(* Structure page *)
	T_ConfigPage:ST_CONFIGPAGE;
	wMaskBtPanelLeft: WORD;
	wMaskBtPanelRight: WORD;
	wMaskFunctionPanel: WORD;
	RisingEdgeProcessDone: R_TRIG;
	xStopImmediatly: BOOL;
	RisingEdgeProcessError: R_TRIG;
	RisingEdgeResetProcess: R_TRIG;
	RisingEdgeExecuteProcess: R_TRIG;
	RisingEdgeActionNotReady: R_TRIG;
	FallingEdgeActionNotReady: F_TRIG;
	RisingEdgeActionDone: R_TRIG;
	xBlockConfirmMessage: BOOL;
	RisingEdgeActionError: R_TRIG;
	RisingEdgeResetAction: R_TRIG;
	xSlowFast: BOOL;
	iSelectedAxis: INT;
	xSlowFastJogToolRotation: BOOL;
	xSlowFastJogToolFeeder: BOOL;
	xSlowFastJogGrindFeeder: BOOL;
	xToggleAxisPower: BOOL;
	xResetAxis: BOOL;
	xUpdateProfileList: BOOL;
	jj: INT;
	RisingEdgePtrProfileListUpDown: R_TRIG;
	iPointerListProfile: INT;
	iActualActiveProfile: INT;
	xAction_CopyProfileToProcess: BOOL;
	xProfileFileNotFound: BOOL;
	iToLoadProfileNr: INT;
	sToLoadProfileName: STRING;
	sTmpDynamicText: STRING;
	xAction_LoadProfileToProcessImage: BOOL;
	xAction_SaveNovRAM: BOOL;
	xActionDeleteProfile: BOOL;
	TimerONTmp: TON;
	iStepActionNovRam: INT;
	xAction_SaveProfileToFile: BOOL;
	iTmp: INT;
	sTmp: STRING;
	sTmp_2: STRING;
	RisingEdgeTimeOut: R_TRIG;
	fbCompareProfileProcessValue:FB_COMPAREPROFILEPROCESSVALUE;
	FailingEdgeGeometryManagement: F_TRIG;
	FailingEdgePrisma: F_TRIG;
	rCalcMinMaxToolDia: REAL;
	xResetParaListValue: BOOL;
	xActivateStationFunction: BOOL;
	iTmpStationFunctionNr: INT;
	xFirstReadInit: BOOL;
	xFirstReadReset: BOOL;
	xMicroRodActive: BOOL;
	FBCalcTorqueToolLeft: FB_CALC_TORQUE;
	FBCalcTorqueToolCenter: FB_CALC_TORQUE;
	FBCalcTorqueToolRight: FB_CALC_TORQUE;
	xTmpStopAxis: BOOL;
	RisingEdgeStartButton: R_TRIG;
	dwPageNrProcessStart: DWORD;
	FallingEdgeStartButton: F_TRIG;
	RisingEdgeStopButton: R_TRIG;
	FallingEdgeStopButton: F_TRIG;
	xToggleCylinderState: BOOL;
	dwTmpActualPage: DWORD;
	xUpdateErrorList: BOOL;
	RisingEdgeErrorList: R_TRIG;
	xParameterSavedErrorList: BOOL;
	xDeleteErrorList: BOOL;
	FBQVisErrorList: FBQVIS_ERROR_LIST;
	FBSetErrorList:FB_SETERRORLIST;
	xProcessMachine: BOOL;
	xProcessStation: BOOL;
	iStepProcess: INT;
	xStepProcessDone: BOOL;
	xStopProcess: BOOL;
	xAction_StopCycle: BOOL;
	xWaitStopEnd: BOOL;
	xWaitStopCycleEnd: BOOL;
	iStepWaitStopEnd: INT;
	xActionProcStation: BOOL;
	xActionProcMachine: BOOL;
	RisingEdgeKeySwitch1: R_TRIG;
	FailingEdgeKeySwitch1: F_TRIG;
	TimerDisplayMessage: TON;
	RisingEdgeReleaseWarning: R_TRIG;
	rCalcPrismaFactor: REAL;
	xFirstReadParaList: BOOL;
	iTmpSelectParaList: INT;
	xAction_SaveNovRAMWithoutConfirm: BOOL;
	diErrorNr: DINT;
	FBErrorMessage : FB_ErrorMessage;
	fbQvisClearError:FBQVIS_CLEARERROR;
	xResetError: BOOL;
	TONTimeWaitMsg: TON;
	xCheckQuitError: BOOL;
	bStateMachine: BYTE;
	xSetStateMachine: BOOL;
	iSelectAxisToolRotation: INT;
	rAutoTimeTotal: REAL;
	rToolRotationSpeed: REAL;
	iAutoProcess: INT;
	xBlockGrindFeederActivation: BOOL;
	xToolFeederMoveStartPos: BOOL;
	xToggleAllAxisPower: BOOL;
	FBCalcProcessTime: FB_CALCPROCESSTIME;
	xReferenceAxis: BOOL;
	xTeachPosition: BOOL;
	xCalcAngleRefIndex: BOOL;
	uiToolLeftZeroTorque: UINT;
	uiToolCenterZeroTorque: UINT;
	uiToolRightZeroTorque: UINT;
	xSetCalculToolRotTorque: BOOL;
	rActualToolFeederPosition: REAL;
	xReadActualToolFeedPos: BOOL;
	xReadActualToolFeedPos1: BOOL;
	rActualToolFeederPosition1: REAL;
	rToolTotalLength: REAL;
	xCalcFirstTime: BOOL;
	xFirstReadParaList1: BOOL;
	iTmpSelectParaList1: INT;
	xTmpTeach: BOOL;
	wTmpActivBtRight: WORD;
	xOverlayGrindFeedSetPlung: BOOL;
	xOpenMessageBox: BOOL;
	lrActualGrindFeedPosition: LREAL;
	lrToWriteGrindFeedPosition: LREAL;
	xCalcAgainProcTime: BOOL;
	xToolFeederMoveLoadPos: BOOL;
	xWarmUp:BOOL;
	iSelectedCylinder: INT;
	xWarmUpMessage: BOOL;
	xWarmUpMessageActiv: BOOL;
	xWarmUpMessageDone: BOOL;
END_VAR
(****************************************************************************************************************************************************)
(******    This Functionblock manage the hole visualisation, it is the interface from the QVis and the control application          *******)
(****************************************************************************************************************************************************)
	IF NOT(xFirstRead) THEN
		xFirstRead:=TRUE;
		T_Visu.ptrT_ExchgParam:=ADR(T_ExchgParam);
	END_IF;
	RisingEdgeActiv(CLK:=T_Visu.T_CtrleVisu.xActive);
	IF RisingEdgeActiv.Q THEN
		(* call functionblock init. *)
		fbQvisInitPage(T_Visu:=T_Visu);
		(* Init. variable for visualisation action *)
		T_Visu.T_CtrleAction.xDone:=TRUE;
		T_Visu.T_CtrleAction.xExecute:=FALSE;
		T_Visu.T_CtrleAction.xNotReady:=FALSE;
		T_Visu.T_CtrleAction.xErr:=FALSE;
		T_Visu.T_CtrleAction.udiErrorID:=0;
		T_Visu.T_CtrleVisu.xDone:=FALSE;
		T_Visu.ptrT_ExchgParam:=ADR(T_ExchgParam);
		wNormalLayerActivTask:=1;
		wSpecialLayerGeneralActivTask:=1;
		wSpecialLayerToolRotActivTask:=1;
		wSpecialLayerWireFeedActivTask:=1;
		wSpecialLayerGrindAxisActivTask:=1;
		wNormalLayerActivPage:=10;
		wSpecialLayerGeneralActivPage:=110;
		wSpecialLayerToolRotActivPage:=210;
		wSpecialLayerWireFeedActivPage:=310;
		wSpecialLayerGrindAxisActivPage:=410;
		T_Visu.ptrT_ExchgParam^.T_TouchScreenNavPanel.wState:=1;
		wStandardPageNr:=10;
		T_Visu.ptrT_ExchgParam^.T_Visu.T_Level.iPwSystem:=999;
		wTmpNormalLayerActivTask:=1;
		wTmpSpecialLayerGeneralActivTask:=1;
		wTmpSpecialLayerToolRotActivTask:=1;
		wTmpSpecialLayerWireFeedActivTask:=1;
		wTmpSpecialLayerGrindAxisActivTask:=1;
		FOR ii:=1 TO 6 DO
			awNormalLayerActivPage[ii]:=wStandardPageNr;
			wStandardPageNr:=wStandardPageNr + 10;
		END_FOR;
		wStandardPageNr:=110;
		FOR ii:=1 TO 6 DO
			awSpecialLayerGeneralActivPage[ii]:=wStandardPageNr;
			wStandardPageNr:=wStandardPageNr + 10;
		END_FOR;
		wStandardPageNr:=210;
		FOR ii:=1 TO 6 DO
			awSpecialLayerToolRotActivPage[ii]:=wStandardPageNr;
			wStandardPageNr:=wStandardPageNr + 10;
		END_FOR;
		wStandardPageNr:=310;
		FOR ii:=1 TO 6 DO
			awSpecialLayerWireFeedActivPage[ii]:=wStandardPageNr;
			wStandardPageNr:=wStandardPageNr + 10;
		END_FOR;
		wStandardPageNr:=410;
		FOR ii:=1 TO 6 DO
			awSpecialLayerGrindAxisActivPage[ii]:=wStandardPageNr;
			wStandardPageNr:=wStandardPageNr + 10;
		END_FOR;
		IF NOT(xFirstReadInit) THEN
			xFirstReadInit:=TRUE;
			T_Visu.T_PlcParam.dwSetNewPage:=1001;
		ELSE
			T_Visu.T_PlcParam.dwSetNewPage:=0;
		END_IF;
		T_Visu.T_PlcParam.dwActualPage:=0;
		T_Visu.T_PlcParam.dwPreviousPage:=0;
		iPointerListProfile:=1;
		iActualActiveProfile:=-1;
		TimerAction(IN:=FALSE);
		(* Init FB *)
		fbQvisClearError(	xExecute:=FALSE,
						iError:=0,
						T_Message:=T_ExchgParam.T_Visu.T_Message,
						T_Station:=T_Station,
						T_Process:=T_Process,
						T_NovRAM:=T_NovRAM,
						T_Profile:=T_Profile,
						T_HDD:=T_HDD,
						xDone=>T_Visu.T_CtrleAction.xDone,
						xNotReady=>T_Visu.T_CtrleAction.xNotReady,
						xErr=>T_Visu.T_CtrleAction.xErr,
						udiErrorID=>T_Visu.T_CtrleAction.udiErrorID);
		T_Visu.ptrT_ExchgParam^.T_Cylinder.iSelectToolTensionForce:=1;	(* For starting the machine set always the process force for the ToolTension *)
		ptrTeachINAxis:=ADR(T_Station.THardware.TAxisToolLeft);
	END_IF;

	IF NOT(T_Visu.T_CtrleVisu.xActive) THEN
		RETURN;
	END_IF;

(* waiting for reset *)
	RisingEdgeReset(CLK:=T_Visu.T_CtrleVisu.xReset);
	IF RisingEdgeReset.Q THEN
		(* Init. structure *)
		T_Visu.T_CtrleVisu.xDone:=FALSE;
		T_Visu.T_CtrleVisu.iFunction:=0;
		T_Visu.T_CtrleVisu.xErr:=FALSE;
		T_Visu.T_CtrleVisu.udiErrorID:=0;
		IF NOT(xFirstReadReset) THEN
			xFirstReadReset:=TRUE;
			T_Visu.T_PlcParam.dwSetNewPage:=1001;
		ELSE
			T_Visu.T_PlcParam.dwSetNewPage:=0;
		END_IF;
		T_Visu.T_PlcParam.dwActualPage:=0;
		T_Visu.T_PlcParam.dwPreviousPage:=0;
		T_Visu.ptrT_ExchgParam^.T_Visu.iQVisActivNewPage:=0;
		wNormalLayerActivTask:=1;
		wSpecialLayerGeneralActivTask:=1;
		wSpecialLayerToolRotActivTask:=1;
		wSpecialLayerWireFeedActivTask:=1;
		wSpecialLayerGrindAxisActivTask:=1;
		wNormalLayerActivPage:=10;
		wSpecialLayerGeneralActivPage:=110;
		wSpecialLayerToolRotActivPage:=210;
		wSpecialLayerWireFeedActivPage:=310;
		wSpecialLayerGrindAxisActivPage:=410;
		wTmpNormalLayerActivTask:=1;
		wTmpSpecialLayerGeneralActivTask:=1;
		wTmpSpecialLayerToolRotActivTask:=1;
		wTmpSpecialLayerWireFeedActivTask:=1;
		wTmpSpecialLayerGrindAxisActivTask:=1;
		T_Visu.ptrT_ExchgParam^.T_TouchScreenNavPanel.wState:=1;
		T_Visu.ptrT_ExchgParam^.T_Visu.bActivSpecialLayer:=0;
		T_Visu.ptrT_ExchgParam^.T_TouchScreenBtPanel.iStateBtLeft:=0;
		wStandardPageNr:=10;
		T_Visu.ptrT_ExchgParam^.T_Visu.T_Level.iPwSystem:=999;
		FOR ii:=1 TO 6 DO
			awNormalLayerActivPage[ii]:=wStandardPageNr;
			wStandardPageNr:=wStandardPageNr + 10;
		END_FOR;
		wStandardPageNr:=110;
		FOR ii:=1 TO 6 DO
			awSpecialLayerGeneralActivPage[ii]:=wStandardPageNr;
			wStandardPageNr:=wStandardPageNr + 10;
		END_FOR;
		wStandardPageNr:=210;
		FOR ii:=1 TO 6 DO
			awSpecialLayerToolRotActivPage[ii]:=wStandardPageNr;
			wStandardPageNr:=wStandardPageNr + 10;
		END_FOR;
		wStandardPageNr:=310;
		FOR ii:=1 TO 6 DO
			awSpecialLayerWireFeedActivPage[ii]:=wStandardPageNr;
			wStandardPageNr:=wStandardPageNr + 10;
		END_FOR;
		wStandardPageNr:=410;
		FOR ii:=1 TO 6 DO
			awSpecialLayerGrindAxisActivPage[ii]:=wStandardPageNr;
			wStandardPageNr:=wStandardPageNr + 10;
		END_FOR;
		(* Activ reset structure control action *)
		T_Visu.T_CtrleAction.xReset:=TRUE;
		(* Activ reset structure control process *)
		T_Visu.T_CtrleProcess.xReset:=TRUE;
		(* Init. pw value *)
		T_Visu.ptrT_ExchgParam^.T_Visu.T_Level.iPwSystem:=999;
		(* Init. Error *)
		T_Visu.ptrT_ExchgParam^.T_Visu.T_Message.iState:=0;
		T_Visu.ptrT_ExchgParam^.T_Visu.T_Message.sDynamicTextEnglish:='';
		T_Visu.ptrT_ExchgParam^.T_Visu.T_Message.sDynamicTextDeutsch:='';
		T_Visu.ptrT_ExchgParam^.T_Visu.T_Message.sDynamicTextFrancais:='';
		T_Visu.ptrT_ExchgParam^.T_TouchScreenBtPanel.iStateBtLeft:=0;
		T_Visu.ptrT_ExchgParam^.T_Cylinder.iSelectCylinder_Sonder1:=1;
		T_Visu.ptrT_ExchgParam^.T_StationCommon.iWireFeederAngleRefIndex:=0;
		T_Visu.ptrT_ExchgParam^.T_TeachIn.iSelectAxisGrind:=1;
		T_Visu.ptrT_ExchgParam^.T_TeachIn.iSelectAxisToolRotation:=1;
		T_Visu.ptrT_ExchgParam^.T_TeachIn.iSelectAxisWireFeeder:=1;
		T_Visu.ptrT_ExchgParam^.T_TeachIn.xSlowFastToolRotation:=FALSE;
		T_Visu.ptrT_ExchgParam^.T_TeachIn.xSlowFastToolFeed:=FALSE;
		T_Visu.ptrT_ExchgParam^.T_TeachIn.xSlowFastGrindFeeder:=FALSE;
		T_Visu.ptrT_ExchgParam^.T_InfoValueCommon.rToolTensionForce:=T_NovRAM.T_Data.T_ProcessImageData.T_ProcessPara.rToolTensionProcess;
		(* active confirmation *)
		xConfirmResetFB:=TRUE;
		(* exit function bloc *)
		RETURN;
	ELSE
		IF xConfirmResetFB THEN
			(* confirm reset FB *)
			T_Visu.T_CtrleVisu.xDone:=TRUE;
			T_Visu.T_CtrleVisu.xErr:=FALSE;
			T_Visu.T_CtrleVisu.udiErrorID:=0;
			(* reset variable *)
			xConfirmResetFB:=FALSE;
			(* activ research if Qvis is activ *)
			xQvisActiv:=TRUE;
			T_Visu.T_CtrleVisu.xQvis:=FALSE;
			dwInCount_QVisCmd:=T_CtrleQVis.dwInCount;
		END_IF
	END_IF

(* determin if qvis activ *)
	IF xQvisActiv THEN
		(* timer time off  *)
		TimerQVis(IN:=TRUE,PT:=T#2s);
		IF dwInCount_QVisCmd = T_CtrleQVis.dwInCount THEN
			(* Init. command *)
			T_CtrleQVis.dwInCommand:=1;
			T_CtrleQVis.dwInQVisCtrlAddress:=ADR(T_CtrleQVis);
			T_CtrleQVis.dwInParameterAddress:=ADR(T_Visu.T_PlcParam.dwSetNewPage);
			(* start command *)
			T_CtrleQVis.dwInCount:=T_CtrleQVis.dwInCount+1;
			(* Activ Timer *)
			TimerQVis(IN:=FALSE);
		ELSE
			IF T_CtrleQVis.dwInCount = T_CtrleQVis.dwOutCount THEN
			(* command done *)
				IF T_CtrleQVis.diOutStatus = 0 THEN
				(* command done without error *)
					xQvisActiv:=FALSE;
					T_Visu.T_CtrleVisu.xQvis:=TRUE;
					T_Visu.T_PlcParam.dwActualPage:=T_Visu.T_PlcParam.dwSetNewPage;
				END_IF
			ELSE
			(* test time off, restart command *)
				IF TimerQVis.Q THEN
					dwInCount_QVisCmd:=T_CtrleQVis.dwInCount;
				END_IF
			END_IF
		END_IF
	END_IF

(* exit FB if Qvis inactiv *)
	IF NOT(T_Visu.T_CtrleVisu.xQvis) THEN RETURN; END_IF

	IF (T_Visu.T_PlcParam.dwActualPage > 0) AND (T_Visu.T_PlcParam.dwActualPage <= 999) THEN
		(* copy config page structure *)
		T_ConfigPage:=T_Visu.T_ConfigPage[T_Visu.T_PageIndex[T_Visu.T_PlcParam.dwActualPage].iIndexConfigPage];
		T_Visu.ptrT_ExchgParam^. T_TouchScreenNavPanel.wNotMasktext:=T_ConfigPage.wMaskTouchScreenNavPanel;
		T_Visu.ptrT_ExchgParam^.T_TouchScreenBtPanel.iNotMaskTextBt:=16#0;
		T_Visu.ptrT_ExchgParam^.T_TouchScreenBtPanel.iNotMaskTextBt:=WORD_TO_INT(INT_TO_WORD(T_Visu.ptrT_ExchgParam^.T_TouchScreenBtPanel.iNotMaskTextBt) OR T_ConfigPage.wMaskBtPanelRight);
		T_Visu.ptrT_ExchgParam^.T_TouchScreenBtPanel.iNotMaskTextBt:=WORD_TO_INT(INT_TO_WORD(T_Visu.ptrT_ExchgParam^.T_TouchScreenBtPanel.iNotMaskTextBt) OR T_ConfigPage.wMaskBtPanelLeft);
		T_Visu.ptrT_ExchgParam^.T_TouchScreenBtPanel.iNotMaskTextBt:=WORD_TO_INT(NOT(INT_TO_WORD(T_Visu.ptrT_ExchgParam^.T_TouchScreenBtPanel.iNotMaskTextBt)));
	END_IF;

(* monitor page Errorlist for Machine *)
	xTmp:=	(T_Visu.T_PlcParam.dwActualPage = 60) OR
			(T_Visu.T_PlcParam.dwActualPage = 160) OR
			(T_Visu.T_PlcParam.dwActualPage = 260) OR
			(T_Visu.T_PlcParam.dwActualPage = 360) OR
			(T_Visu.T_PlcParam.dwActualPage = 460);
	IF xTmp THEN
		(* Check if Station will be changed without change the Error Page *)
		IF (dwTmpActualPage <> T_Visu.T_PlcParam.dwActualPage) THEN
			xUpdateErrorList:=TRUE;
			dwTmpActualPage:=T_Visu.T_PlcParam.dwActualPage;
		END_IF;
	END_IF;
	IF xTmp OR xUpdateErrorList THEN
		IF NOT(xTmp) AND xUpdateErrorList THEN
			RisingEdgeErrorList(CLK:=xUpdateErrorList);
		ELSE
			RisingEdgeErrorList(CLK:=xTmp AND NOT(xUpdateErrorList));
		END_IF;
		xUpdateErrorList:=FALSE;
		IF RisingEdgeErrorList.Q THEN
			FBQVisErrorList(	T_ErrorList:= T_ErrorList,
							T_ErrorNrList:= T_NovRAM.T_Data.T_ErrorNrList,
							T_MsgErrorEnglish:= T_Visu.ptrT_ExchgParam^.T_Visu.T_MsgErrorEnglish,
							T_MsgErrorDeutsch:= T_Visu.ptrT_ExchgParam^.T_Visu.T_MsgErrorDeutsch,
							T_MsgErrorFrancais:= T_Visu.ptrT_ExchgParam^.T_Visu.T_MsgErrorFrancais);
		END_IF;
	ELSE
		RisingEdgeErrorList(CLK:=FALSE);
	END_IF;

(* Refresh Errorlist for Machine and Station *)
	FBSetErrorList(	TControlStation:= T_Station.TControl,
					TProcess:= T_Process,
					xParameterSaved:= xParameterSavedErrorList,
					T_ErrorNrList:= T_NovRAM.T_Data.T_ErrorNrList,
					xSetForceError:= T_Visu.ptrT_ExchgParam^.T_SafetyCtrl.xSetForceError,
					diSetForceErrorNr:= T_Visu.ptrT_ExchgParam^.T_SafetyCtrl.diSetForceErrorNr);
	IF FBSetErrorList.xSaveParameter THEN
		IF T_Visu.T_CtrleAction.xDone AND NOT(T_Visu.T_CtrleAction.xExecute) AND T_NovRAM.T_Ctrle.xDone AND NOT(T_NovRAM.T_Ctrle.xExecute) THEN
			xParameterSavedErrorList:=TRUE;
			xUpdateErrorList:=TRUE;
			T_NovRAM.T_Ctrle.xExecute:=TRUE;
			T_NovRAM.T_Ctrle.iFunction:=2;
			T_NovRAM.T_Data.T_ErrorNrList;
		END_IF;
	END_IF;

(* Monitoring Visu Parameter *)
	T_Visu.ptrT_ExchgParam^.T_StationCommon.rConvertMaxToolLength:=T_NovRAM.T_Data.T_Standard.T_MachineConfig.rConfigMaxToolLength * 10.0;	(* convert from cm to mm *)
	T_Visu.ptrT_ExchgParam^.T_StationCommon.T_ParamToolTensionSystem.rMaxForceTT:=T_NovRAM.T_Data.T_Standard.T_ToolTensionSystem.rMaxForceTT;
	IF (T_NovRam.T_Data.T_Standard.T_MachineConfig.iConfigMachineType = 2) THEN
		xMicroRodActive:=TRUE;
	ELSE
		xMicroRodActive:=FALSE;
	END_IF;
	IF (T_Visu.T_PlcParam.dwActualPage = 170) AND ((T_Visu.ptrT_ExchgParam^.T_Config.iEditParam >= 120) AND (T_Visu.ptrT_ExchgParam^.T_Config.iEditParam <= 129)) THEN
		IF NOT(xFirstReadParaList) THEN
			iTmpSelectParaList:=T_Visu.ptrT_ExchgParam^.T_Config.iSelectParaList;
		END_IF;
		xFirstReadParaList:=TRUE;
		T_Visu.ptrT_ExchgParam^.T_Config.xBlockParaListNavi:=FALSE;
		T_Visu.ptrT_ExchgParam^.T_Config.xBlockParaListNavi1:=TRUE;
		T_Visu.ptrT_ExchgParam^.T_Config.xBlockProfilList:=FALSE;
		T_Visu.ptrT_ExchgParam^.T_Config.xBlockNavParaList:=FALSE;
		T_Visu.ptrT_ExchgParam^.T_Config.iEditParam:=iFctGetEditParaList(	dwActualPage:=120,
																	xMicroRodActive:=xMicroRodActive,
																	iSelectParaList:=T_Visu.ptrT_ExchgParam^.T_Config.iSelectParaList,
																	iSelectParaListTeachRot:=T_Visu.ptrT_ExchgParam^.T_Config.iSelectParaListTeachRot);
		(* 09.12.2010 KFS:	{	*)
		IF (T_ExchgParam.T_Visu.T_Level.iActLevel <>2) THEN
			IF  (T_Visu.ptrT_ExchgParam^.T_Config.iEditParam = 121) THEN
				 T_Visu.ptrT_ExchgParam^.T_Config.iEditParam:= 126;
			ELSIF ( T_Visu.ptrT_ExchgParam^.T_Config.iEditParam = 123) THEN
				 T_Visu.ptrT_ExchgParam^.T_Config.iEditParam:= 127;
			ELSIF ( T_Visu.ptrT_ExchgParam^.T_Config.iEditParam = 125) THEN
				 T_Visu.ptrT_ExchgParam^.T_Config.iEditParam:= 128;
			END_IF;
		END_IF;
		(* 09.12.2010 KFS:	}	*)
		IF (iTmpSelectParaList <> T_Visu.ptrT_ExchgParam^.T_Config.iSelectParaList) THEN
			iTmpSelectParaList:=T_Visu.ptrT_ExchgParam^.T_Config.iSelectParaList;
			xResetParaListValue:=TRUE;
		END_IF;
	ELSE
		xFirstReadParaList:=FALSE;
		T_Visu.ptrT_ExchgParam^.T_Config.xBlockNavParaList:=TRUE;
	END_IF;
	IF (T_Visu.T_PlcParam.dwActualPage = 270) AND ((T_Visu.ptrT_ExchgParam^.T_Config.iEditParam >= 210) AND (T_Visu.ptrT_ExchgParam^.T_Config.iEditParam <= 219)) THEN
		IF NOT(xFirstReadParaList1) THEN
			iTmpSelectParaList1:=T_Visu.ptrT_ExchgParam^.T_Config.iSelectParaListTeachRot;
		END_IF;
		xFirstReadParaList1:=TRUE;
		T_Visu.ptrT_ExchgParam^.T_Config.xBlockNavParaListTeachRot:=FALSE;
		T_Visu.ptrT_ExchgParam^.T_Config.iEditParam:=iFctGetEditParaList(	dwActualPage:=210,
																	xMicroRodActive:=xMicroRodActive,
																	iSelectParaList:=T_Visu.ptrT_ExchgParam^.T_Config.iSelectParaListTeachRot,
																	iSelectParaListTeachRot:=T_Visu.ptrT_ExchgParam^.T_Config.iSelectParaListTeachRot);
		IF (iTmpSelectParaList1 <> T_Visu.ptrT_ExchgParam^.T_Config.iSelectParaListTeachRot) THEN
			iTmpSelectParaList1:=T_Visu.ptrT_ExchgParam^.T_Config.iSelectParaListTeachRot;
			xResetParaListValue:=TRUE;
		END_IF;
	ELSE
		xFirstReadParaList1:=FALSE;
		T_Visu.ptrT_ExchgParam^.T_Config.xBlockNavParaListTeachRot:=TRUE;
	END_IF;
	xTmp:=	(T_Visu.T_PlcParam.dwActualPage = 170) OR
			(T_Visu.T_PlcParam.dwActualPage = 270) OR
			(T_Visu.T_PlcParam.dwActualPage = 370) OR
			(T_Visu.T_PlcParam.dwActualPage = 470);
	IF xTmp AND (T_Visu.ptrT_ExchgParam^.T_Config.iEditParam = 0) THEN
		T_Visu.ptrT_ExchgParam^.T_Config.xBlockParaListNavi:=TRUE;
		T_Visu.ptrT_ExchgParam^.T_Config.xBlockParaListNavi1:=TRUE;
	END_IF;

(* Monitor dynamic mask for button panel left and right and function panel *)
	IF T_Visu.T_CtrleProcess.xDone OR T_Visu.T_CtrleProcess.xErr THEN
	(* Set the standard mask *)
		wMaskBtPanelLeft:=T_ConfigPage.wMaskBtPanelLeft;
		wMaskBtPanelRight:=T_ConfigPage.wMaskBtPanelRight;
		wMaskFunctionPanel:=T_ConfigPage.wMaskFunctionPanel;
	(* Set the dynamic mask *)
	ELSE	wMaskBtPanelLeft:=T_ConfigPage.wMaskBtPanelLeft AND T_ConfigPage.wMaskActiveMachineBtPanelLeft;
			wMaskBtPanelRight:=T_ConfigPage.wMaskActiveMachineBtPanelRight;
			wMaskFunctionPanel:=T_ConfigPage.wMaskActiveMachineFunctionPanel;
	END_IF
	(* Check activ Page *)
	IF (T_Visu.T_PlcParam.dwActualPage = 170) OR (T_Visu.T_PlcParam.dwActualPage = 270) OR (T_Visu.T_PlcParam.dwActualPage = 370) OR (T_Visu.T_PlcParam.dwActualPage = 470) THEN
		IF (T_Visu.ptrT_ExchgParam^.T_Config.iEditParam = 0) THEN
			wMaskBtPanelRight:=16#0;
		END_IF;
		IF (T_Visu.ptrT_ExchgParam^.T_Config.iEditParam = 130) OR (T_Visu.ptrT_ExchgParam^.T_Config.iEditParam = 131) THEN
			wMaskBtPanelRight:=16#0;
		END_IF;
	END_IF;
	(* Config. divers mask *)
	T_Visu.ptrT_ExchgParam^.T_TouchScreenBtPanel.iNotMaskTextBt
		:=(16#1F XOR wMaskBtPanelLeft) OR (16#3E0 XOR wMaskBtPanelRight);
	(* management Fn button panel availability *)
	T_Visu.ptrT_ExchgParam^.T_BtFunctionPanel.wNotMasktext:=16#FFF XOR wMaskFunctionPanel;
	(* management navigation panel mask *)
	T_Visu.ptrT_ExchgParam^.T_TouchScreenNavPanel.wNotMasktext:=T_ConfigPage.wMaskTouchScreenNavPanel;

(************************************************************************************************************************************************************************)
(********start of the managment of the external start-stop button, special button and function button and task button and external tool buttons********)
(************************************************************************************************************************************************************************)
(* Start button *)
	(* ...manage action button *)
	xTmp:=	NOT(xChangePage)
			AND (T_Visu.T_CtrleAction.xDone)
			AND NOT(T_Visu.T_CtrleAction.xExecute);
	IF xTmp THEN
		(* manage rising edge start button *)
		RisingEdgeStartButton(CLK:=xStartButton AND T_ConfigPage.xMaskBtStart);
		IF RisingEdgeStartButton.Q AND bButtonPanelLocked = 16#0 AND NOT(T_StartUp.T_State.xBlockChangeMovementVisu) THEN
		(* panel locked *)
			bButtonPanelLocked:=16#10;
			(* Start process at the begin *)
			T_Visu.T_CtrleAction.xExecute:=TRUE;
			CASE T_Visu.T_PlcParam.dwActualPage OF
			(* Data machine *)
			10:	T_Visu.T_CtrleAction.iFunction:=710;
			20:	T_Visu.T_CtrleAction.iFunction:=720;
			30:	T_Visu.T_CtrleAction.iFunction:=730;
			110:	T_Visu.T_CtrleAction.iFunction:=640;
			210:	T_Visu.T_CtrleAction.iFunction:=318;
			220:	T_Visu.T_CtrleAction.iFunction:=402;
			310:	T_Visu.T_CtrleAction.iFunction:=305;
			330:	T_Visu.T_CtrleAction.iFunction:=420;
			410:	T_Visu.T_CtrleAction.iFunction:=305;
			ELSE
				T_Visu.T_CtrleAction.xExecute:=FALSE;
			END_CASE
			(* save page number for stop procedure *)
			IF T_Visu.T_CtrleAction.xExecute THEN
				dwPageNrProcessStart:=T_Visu.T_PlcParam.dwActualPage;
				xStopImmediatly:=FALSE;
			END_IF
		END_IF
		(* manage falling edge start button *)
		FallingEdgeStartButton(CLK:=xStartButton AND T_ConfigPage.xMaskBtStart);
		IF FallingEdgeStartButton.Q AND (bButtonPanelLocked AND 16#10) = 16#10 THEN bButtonPanelLocked:=bButtonPanelLocked XOR 16#10; END_IF
	ELSE
		RisingEdgeStartButton(CLK:=FALSE);
		FallingEdgeStartButton(CLK:=TRUE);
	END_IF

(* Stop button *)
	xTmp:=	NOT(T_Visu.T_CtrleAction.xExecute);
	xTmpTeach:=((T_Visu.T_PlcParam.dwActualPage = 310) OR (T_Visu.T_PlcParam.dwActualPage = 410)) AND (bButtonPanelLocked = 16#10);
	IF xTmp THEN
		RisingEdgeStopButton(CLK:=xStopButton);
		IF RisingEdgeStopButton.Q AND ((bButtonPanelLocked = 16#0) OR xTmpTeach) THEN
		(* pane locked *)
			bButtonPanelLocked:=16#20;
			(* activ stop process *)
			T_Visu.T_CtrleAction.xExecute:=TRUE;
			CASE T_Visu.T_PlcParam.dwActualPage OF
			10:	T_Visu.T_CtrleAction.iFunction:=800;
			20:	T_Visu.T_CtrleAction.iFunction:=800;
			30:	T_Visu.T_CtrleAction.iFunction:=800;
			110:	T_Visu.T_CtrleAction.iFunction:=800;
				T_Visu.ptrT_ExchgParam^.T_Visu.T_Message.iState:=121;
			210:	T_Visu.T_CtrleAction.iFunction:=301;
				T_Visu.ptrT_ExchgParam^.T_Visu.T_Message.iState:=121;
			220:	T_Visu.T_CtrleAction.iFunction:=403;
				T_Visu.ptrT_ExchgParam^.T_Visu.T_Message.iState:=121;
			310:	T_Visu.T_CtrleAction.iFunction:=301;
				T_Visu.ptrT_ExchgParam^.T_Visu.T_Message.iState:=121;
			330:	T_Visu.T_CtrleAction.iFunction:=800;
				T_Visu.ptrT_ExchgParam^.T_Visu.T_Message.iState:=121;
			410:	T_Visu.T_CtrleAction.iFunction:=301;
				T_Visu.ptrT_ExchgParam^.T_Visu.T_Message.iState:=121;
			ELSE
				T_Visu.T_CtrleAction.xExecute:=FALSE;
			END_CASE
		END_IF
		(* manage falling edge stop button *)
		FallingEdgeStopButton(CLK:=xStopButton AND T_ConfigPage.xMaskBtStop);
		IF FallingEdgeStopButton.Q AND (bButtonPanelLocked AND 16#20) = 16#20 THEN
			bButtonPanelLocked:=bButtonPanelLocked XOR 16#20; END_IF
	ELSE
		RisingEdgeStopButton(CLK:=FALSE);
		FallingEdgeStopButton(CLK:=TRUE);
	END_IF

(* Management Bt Panel left *)
	IF T_Visu.ptrT_ExchgParam^.T_Config.xNoTouchScreenBtPanel THEN
		wActivBtLeft:=wSPSSpecialButton;
	ELSE
		wActivBtLeft:=INT_TO_WORD(T_Visu.ptrT_ExchgParam^.T_TouchScreenBtPanel.iActivBtLeft);
	END_IF;
	RisingEdgeSpecialLayer(CLK:=xSecurityKey);
	FallingEdgeSpecialLayer(CLK:=xSecurityKey);
	RisingEdgeBtPanelLeft(CLK:=((wActivBtLeft AND wMaskBtPanelLeft) <> 16#0) AND T_Visu.ptrT_ExchgParam^.T_Visu.bActivSpecialLayer <> 0);
	FallingEdgeBtPanelLeft(CLK:=((wActivBtLeft AND wMaskBtPanelLeft) <> 16#0) AND T_Visu.ptrT_ExchgParam^.T_Visu.bActivSpecialLayer <> 0);
	xTmp:=	NOT(xChangePage)
			AND (T_Visu.T_CtrleAction.xDone OR ((xOverlayMeasureToolDia OR xOverlayGrindFeedSetPlung OR T_Visu.ptrT_ExchgParam^.T_FunctionCommon.xOpenOverlayMessageBox) AND FallingEdgeSpecialLayer.Q))
			AND NOT(T_Visu.T_CtrleAction.xExecute)
			AND NOT(T_StartUp.T_State.xBlockChangeMovementVisu)
			AND NOT(T_StartUp.T_State.xBlockVisuNavigation)
			AND T_StartUp.T_State.xCompleted;
	IF xTmp THEN
		IF RisingEdgeSpecialLayer.Q THEN
			CASE bOldActivSpecialLayer OF
				1:	T_Visu.ptrT_ExchgParam^.T_Visu.bActivSpecialLayer:=1;
					T_Visu.ptrT_ExchgParam^.T_TouchScreenBtPanel.iStateBtLeft:=1;
					T_Visu.ptrT_ExchgParam^.T_TouchScreenNavPanel.wState:=wSpecialLayerGeneralActivTask;
					ii:=1;
					wTmp:=wSpecialLayerGeneralActivTask;
					WHILE wTmp <> 16#0 DO
						IF (wTmp AND 16#1) = 16#1 THEN EXIT; END_IF
						wTmp:=ROR(wTmp,1);
						ii:=ii+1;
					END_WHILE
					dwSetNewPage:=awSpecialLayerGeneralActivPage[ii];
				2:	T_Visu.ptrT_ExchgParam^.T_Visu.bActivSpecialLayer:=2;
					T_Visu.ptrT_ExchgParam^.T_TouchScreenBtPanel.iStateBtLeft:=2;
					T_Visu.ptrT_ExchgParam^.T_TouchScreenNavPanel.wState:=wSpecialLayerToolRotActivTask;
					ii:=1;
					wTmp:=wSpecialLayerToolRotActivTask;
					WHILE wTmp <> 16#0 DO
						IF (wTmp AND 16#1) = 16#1 THEN EXIT; END_IF
						wTmp:=ROR(wTmp,1);
						ii:=ii+1;
					END_WHILE
					dwSetNewPage:=awSpecialLayerToolRotActivPage[ii];
				3:	T_Visu.ptrT_ExchgParam^.T_Visu.bActivSpecialLayer:=3;
					T_Visu.ptrT_ExchgParam^.T_TouchScreenBtPanel.iStateBtLeft:=4;
					T_Visu.ptrT_ExchgParam^.T_TouchScreenNavPanel.wState:=wSpecialLayerWireFeedActivTask;
					ii:=1;
					wTmp:=wSpecialLayerWireFeedActivTask;
					WHILE wTmp <> 16#0 DO
						IF (wTmp AND 16#1) = 16#1 THEN EXIT; END_IF
						wTmp:=ROR(wTmp,1);
						ii:=ii+1;
					END_WHILE
					dwSetNewPage:=awSpecialLayerWireFeedActivPage[ii];
				4:	T_Visu.ptrT_ExchgParam^.T_Visu.bActivSpecialLayer:=4;
					T_Visu.ptrT_ExchgParam^.T_TouchScreenBtPanel.iStateBtLeft:=8;
					T_Visu.ptrT_ExchgParam^.T_TouchScreenNavPanel.wState:=wSpecialLayerGrindAxisActivTask;
					ii:=1;
					wTmp:=wSpecialLayerGrindAxisActivTask;
					WHILE wTmp <> 16#0 DO
						IF (wTmp AND 16#1) = 16#1 THEN EXIT; END_IF
						wTmp:=ROR(wTmp,1);
						ii:=ii+1;
					END_WHILE
					dwSetNewPage:=awSpecialLayerGrindAxisActivPage[ii];
			ELSE
				T_Visu.ptrT_ExchgParam^.T_Visu.bActivSpecialLayer:=1;
				T_Visu.ptrT_ExchgParam^.T_TouchScreenBtPanel.iStateBtLeft:=1;
				T_Visu.ptrT_ExchgParam^.T_TouchScreenNavPanel.wState:=wSpecialLayerGeneralActivTask;
				dwSetNewPage:=wSpecialLayerGeneralActivPage;
			END_CASE;
			T_Visu.T_CtrleAction.iFunction:=6;
			T_Visu.T_CtrleAction.xExecute:=TRUE;
		END_IF;

		IF FallingEdgeSpecialLayer.Q THEN
			IF xOverlayMeasureToolDia THEN
				T_Visu.ptrT_ExchgParam^.T_FunctionCommon.xOpenOverlayMeasureInput:=FALSE;
				T_Visu.ptrT_ExchgParam^.T_FunctionCommon.xSaveButton:=FALSE;
				T_Visu.ptrT_ExchgParam^.T_FunctionCommon.xExitButton:=FALSE;
				T_Visu.ptrT_ExchgParam^.T_FunctionCommon.xHideProgressbar:=FALSE;
				xOverlayMeasureToolDia:=FALSE;
				T_Visu.T_CtrleAction.xDone:=TRUE;
			END_IF;
			IF xOverlayGrindFeedSetPlung THEN
				T_Visu.ptrT_ExchgParam^.T_FunctionCommon.xOpenOverlaySetGrindPlunge:=FALSE;
				T_Visu.ptrT_ExchgParam^.T_FunctionCommon.xSaveButton:=FALSE;
				T_Visu.ptrT_ExchgParam^.T_FunctionCommon.xExitButton:=FALSE;
				T_Visu.ptrT_ExchgParam^.T_FunctionCommon.xHideProgressbar:=FALSE;
				xOverlayGrindFeedSetPlung:=FALSE;
				T_Visu.T_CtrleAction.xDone:=TRUE;
			END_IF;
			IF T_Visu.ptrT_ExchgParam^.T_FunctionCommon.xOpenOverlayMessageBox THEN
				T_Visu.ptrT_ExchgParam^.T_FunctionCommon.xOpenOverlayMessageBox:=FALSE;
				xAction_SaveNovRAM:=FALSE;
				xAction_SaveNovRAMWithoutConfirm:=FALSE;
			END_IF;
			T_Visu.ptrT_ExchgParam^.T_Visu.bActivSpecialLayer:=0;
			T_Visu.ptrT_ExchgParam^.T_TouchScreenBtPanel.iStateBtLeft:=0;
			T_Visu.ptrT_ExchgParam^.T_TouchScreenNavPanel.wState:=wNormalLayerActivTask;
			ii:=1;
			wTmp:=wNormalLayerActivTask;
			WHILE wTmp <> 16#0 DO
				IF (wTmp AND 16#1) = 16#1 THEN EXIT; END_IF
				wTmp:=ROR(wTmp,1);
				ii:=ii+1;
			END_WHILE
			dwSetNewPage:=awNormalLayerActivPage[ii];
			T_Visu.T_CtrleAction.iFunction:=6;
			T_Visu.T_CtrleAction.xExecute:=TRUE;
		END_IF;
		IF wActivBtLeft = 16#10 THEN
			CASE T_Visu.ptrT_ExchgParam^.T_Visu.bActivSpecialLayer OF
				1:	iTmpActivBtLeft:=1;
				2:	iTmpActivBtLeft:=2;
				3:	iTmpActivBtLeft:=4;
				4:	iTmpActivBtLeft:=8;
			END_CASE;
		ELSE
			iTmpActivBtLeft:=WORD_TO_INT(wActivBtLeft);
		END_IF;
		IF RisingEdgeBtPanelLeft.Q THEN
			iStepCounter:=iStepCounter + 1;
			CASE iTmpActivBtLeft OF
				16#1:	T_Visu.ptrT_ExchgParam^.T_Visu.bActivSpecialLayer:=1;
						T_Visu.ptrT_ExchgParam^.T_TouchScreenNavPanel.wState:=wSpecialLayerGeneralActivTask;
						dwSetNewPage:=wSpecialLayerGeneralActivPage;
				16#2:	T_Visu.ptrT_ExchgParam^.T_Visu.bActivSpecialLayer:=2;
						T_Visu.ptrT_ExchgParam^.T_TouchScreenNavPanel.wState:=wSpecialLayerToolRotActivTask;
						dwSetNewPage:=wSpecialLayerToolRotActivPage;
				16#4:	T_Visu.ptrT_ExchgParam^.T_Visu.bActivSpecialLayer:=3;
						T_Visu.ptrT_ExchgParam^.T_TouchScreenNavPanel.wState:=wSpecialLayerWireFeedActivTask;
						dwSetNewPage:=wSpecialLayerWireFeedActivPage;
				16#8:	T_Visu.ptrT_ExchgParam^.T_Visu.bActivSpecialLayer:=4;
						T_Visu.ptrT_ExchgParam^.T_TouchScreenNavPanel.wState:=wSpecialLayerGrindAxisActivTask;
						dwSetNewPage:=wSpecialLayerGrindAxisActivPage;
			END_CASE;
			bOldActivSpecialLayer:=T_Visu.ptrT_ExchgParam^.T_Visu.bActivSpecialLayer;
			IF ((wActivBtLeft AND 16#10) <> 16#10) THEN
				IF ((INT_TO_WORD(T_Visu.ptrT_ExchgParam^.T_TouchScreenBtPanel.iStateBtLeft) AND 16#10) = 16#10) THEN
					T_Visu.ptrT_ExchgParam^.T_TouchScreenBtPanel.iStateBtLeft:=WORD_TO_INT(wActivBtLeft OR 16#10);
					T_Visu.T_CtrleAction.iFunction:=3;
					T_Visu.T_CtrleAction.xExecute:=TRUE;
					xResetParaListValue:=TRUE;
				ELSE
					T_Visu.ptrT_ExchgParam^.T_TouchScreenBtPanel.iStateBtLeft:=WORD_TO_INT(wActivBtLeft);
					T_Visu.T_CtrleAction.iFunction:=6;
					T_Visu.T_CtrleAction.xExecute:=TRUE;
				END_IF;
			ELSE
				IF ((INT_TO_WORD(T_Visu.ptrT_ExchgParam^.T_TouchScreenBtPanel.iStateBtLeft) AND 16#10) = 16#10) THEN
					T_Visu.ptrT_ExchgParam^.T_TouchScreenBtPanel.iStateBtLeft:=T_Visu.ptrT_ExchgParam^.T_TouchScreenBtPanel.iStateBtLeft - 16#10;
					T_Visu.T_CtrleAction.iFunction:=6;
					T_Visu.T_CtrleAction.xExecute:=TRUE;
					xResetParaListValue:=TRUE;
				ELSE
					T_Visu.ptrT_ExchgParam^.T_TouchScreenBtPanel.iStateBtLeft:=WORD_TO_INT(wActivBtLeft OR INT_TO_WORD(T_Visu.ptrT_ExchgParam^.T_TouchScreenBtPanel.iStateBtLeft));
					T_Visu.T_CtrleAction.iFunction:=3;
					T_Visu.T_CtrleAction.xExecute:=TRUE;
					xResetParaListValue:=TRUE;
				END_IF;
			END_IF;
		END_IF;
	END_IF;

(* Management Bt Panel Right *)
	IF (T_Visu.T_PlcParam.dwActualPage = 320) THEN
		IF NOT(xMicroRodActive) THEN
		(* For MicroWire no Function for ToolFeeder-->Cancel Function F1, F2, F3 and F4 *)
			wMaskBtPanelRight:=wMaskBtPanelRight AND 16#0;
			T_Visu.ptrT_ExchgParam^.T_TouchScreenBtPanel.iNotMaskTextBt:=WORD_TO_INT(INT_TO_WORD(T_Visu.ptrT_ExchgParam^.T_TouchScreenBtPanel.iNotMaskTextBt) OR 16#3E0);
		END_IF;
	END_IF;
	IF (T_Visu.T_PlcParam.dwActualPage = 10) THEN
		IF (T_NovRam.T_Data.T_ProcessImageData.T_AutoGeometryPara.iCycleGeometry <= 1) THEN
			T_Visu.ptrT_ExchgParam^.T_TouchScreenBtPanel.iNotMaskTextBt:=WORD_TO_INT(INT_TO_WORD(T_Visu.ptrT_ExchgParam^.T_TouchScreenBtPanel.iNotMaskTextBt) OR 16#1E0);
		END_IF;
	END_IF;
	TimerPressBtPanelRight(IN:=TRUE, PT:=T#3600s);
	IF T_Visu.ptrT_ExchgParam^.T_Config.xNoTouchScreenBtPanel THEN
		wActivBtRight:=wSPSSpecialButton;
	ELSE
		wActivBtRight:=INT_TO_WORD(T_Visu.ptrT_ExchgParam^.T_TouchScreenBtPanel.iActivBtRight);
	END_IF;
	RisingEdgeBtPanelRight(CLK:=(wActivBtRight AND wMaskBtPanelRight) <> 16#0);
	FallingEdgeBtPanelRight(CLK:=(wActivBtRight AND wMaskBtPanelRight) <> 16#0);
	xTmp:=	(NOT(xChangePage)
			AND T_Visu.T_CtrleAction.xDone
			AND NOT(T_Visu.T_CtrleAction.xExecute)
			AND NOT(T_StartUp.T_State.xBlockChangeMovementVisu)
			(*AND NOT(T_StartUp.T_State.xBlockVisuNavigation)*))
			OR xDelayActionBtPanelRight;
	IF (wActivBtRight = 0) AND NOT(xDelayActionBtPanelRight) THEN
		TimerPressBtPanelRight(IN:=FALSE);
	END_IF;
	IF xTmp THEN
		(* Rising edge action *)
		IF RisingEdgeBtPanelRight.Q AND (bButtonPanelLocked = 16#0) AND (NOT(T_StartUp.T_State.xBlockVisuNavigation) OR ((T_NovRam.T_Data.T_ProcessImageData.T_AutoGeometryPara.iCycleGeometry > 1)) AND (T_Visu.T_PlcParam.dwActualPage = 10)) THEN
		(* init. variable *)
			ii:=1;
			wTmp:=wActivBtRight;
			wTmpActivBtRight:=wActivBtRight;
			wTmp:=ROR(wTmp,5);
			(* only one button is used *)
			WHILE wTmp <> 16#0 DO
				IF (wTmp AND 16#1) = 16#1 THEN EXIT; END_IF
				wTmp:=ROR(wTmp,1);
				ii:=ii+1;
			END_WHILE
			(* set the new action if present *)
			IF T_ConfigPage.aiRTrigActionPanelRight[ii] <> 0 THEN
				T_Visu.T_CtrleAction.iFunction:=T_ConfigPage.aiRTrigActionPanelRight[ii];
				T_Visu.T_CtrleAction.xExecute:=TRUE;
			END_IF
			IF (T_ConfigPage.aiFTrigActionPanelRight[ii] = 301) THEN
				xTmpStopAxis:=TRUE;
			END_IF
			(* init. timer press button *)
			TimerPressBtPanelRight(IN:=FALSE);
			(* Lock button panel *)
			bButtonPanelLocked:=16#2;
			(* init. variable *)
			xDelayActionBtPanelRight:=FALSE;
		END_IF
		(* Falling Edge action activ only if the delay action has been started *)
		IF FallingEdgeBtPanelRight.Q AND ((bButtonPanelLocked AND 16#2) = 16#2) THEN
			ii:=1;
			wTmp:=wTmpActivBtRight;
			wTmp:=ROR(wTmp,5);
			(* only one button is used *)
			WHILE wTmp <> 16#0 DO
				IF (wTmp AND 16#1) = 16#1 THEN EXIT; END_IF
				wTmp:=ROR(wTmp,1);
				ii:=ii+1;
			END_WHILE
			(* set the new action if present *)
			IF T_ConfigPage.aiFTrigActionPanelRight[ii] <> 0 (*AND xDelayActionBtPanelRight*) THEN
				T_Visu.T_CtrleAction.iFunction:=T_ConfigPage.aiFTrigActionPanelRight[ii];
				T_Visu.T_CtrleAction.xExecute:=TRUE;
				IF (T_Visu.T_CtrleAction.iFunction = 301) THEN
					xTmpStopAxis:=TRUE;
				END_IF;
			END_IF
			(* release lock panel *)
			bButtonPanelLocked:=bButtonPanelLocked XOR 16#2;
			(* init. variable *)
			xDelayActionBtPanelRight:=FALSE;
		END_IF;

		(* monitor delay *)
		xTmp:=	NOT(xDelayActionBtPanelRight)
				AND NOT(FallingEdgeBtPanelRight.Q)
				AND (bButtonPanelLocked AND 16#2) =16#2;
		IF xTmp AND (TimerPressBtPanelRight.ET > T#500ms) THEN
		(* activ delay action *)
			ii:=1;
			wTmp:=wActivBtRight;
			wTmp:=ROR(wTmp,5);
			(* only one button is used *)
			WHILE wTmp <> 16#0 DO
				IF (wTmp AND 16#1) = 16#1 THEN EXIT; END_IF
				wTmp:=ROR(wTmp,1);
				ii:=ii+1;
			END_WHILE
			(* set the new action if present *)
			IF T_ConfigPage.aiDelayActionPanelRight[ii] <> 0 THEN
				T_Visu.T_CtrleAction.iFunction:=T_ConfigPage.aiDelayActionPanelRight[ii];
				T_Visu.T_CtrleAction.xExecute:=TRUE;
			END_IF
			(* confirm execution delay action *)
			xDelayActionBtPanelRight:=TRUE;
		END_IF;
		IF T_Visu.T_CtrleAction.xDone AND (wActivBtRight = 16#0) AND (bButtonPanelLocked = 16#2) THEN
			bButtonPanelLocked:=0;
		END_IF;
	END_IF
	IF xTmpStopAxis THEN
		IF ptrTeachINAxis^.T_CtrleSingle.xErr THEN
			IF (ptrTeachINAxis^.T_Config_Gen.iTyp <> 0) THEN
				diErrorNr:=(ptrTeachINAxis^.T_Config_Gen.iTyp * 1000000) + ptrTeachINAxis^.T_CtrleSingle.udiErrorID;
			ELSE
				diErrorNr:=0;
			END_IF;
			FBErrorMessage(	diErrorNr:=diErrorNr,
							T_ErrorList:=T_ErrorList);
			T_Visu.ptrT_ExchgParam^.T_Visu.T_Message.sDynamicTextEnglish:=FBErrorMessage.sErrorTextEnglish;
			T_Visu.ptrT_ExchgParam^.T_Visu.T_Message.sDynamicTextDeutsch:=FBErrorMessage.sErrorTextDeutsch;
			T_Visu.ptrT_ExchgParam^.T_Visu.T_Message.sDynamicTextFrancais:=FBErrorMessage.sErrorTextFrancais;
			T_Visu.ptrT_ExchgParam^.T_SafetyCtrl.xSetForceError:=TRUE;
			T_Visu.ptrT_ExchgParam^.T_SafetyCtrl.diSetForceErrorNr:=diErrorNr;
			ptrTeachINAxis^.T_CtrleSingle.iFunction:=1;
			ptrTeachINAxis^.T_CtrleSingle.xExecute:=TRUE;
			T_StartUp.T_Ctrle.xSetSecurityStateON:=TRUE;
		END_IF;
	END_IF;
	IF xTmpStopAxis AND T_Visu.T_CtrleAction.xDone AND (bButtonPanelLocked = 0) AND NOT(T_Visu.T_CtrleAction.xExecute) AND (NOT(T_Station.THardware.TAxisToolLeft.T_CtrleSingle.xNotMoving) OR
	    (NOT(T_Station.THardware.TAxisToolCenter.T_CtrleSingle.xNotMoving) AND xMicroRodActive) OR NOT(T_Station.THardware.TAxisToolRight.T_CtrleSingle.xNotMoving) OR
	     NOT(T_Station.THardware.TAxisToolFeeder.T_CtrleSingle.xNotMoving) OR NOT(T_Station.THardware.TAxisGrindFeeder.T_CtrleSingle.xNotMoving)) THEN
		T_Visu.T_CtrleAction.iFunction:=301;
		T_Visu.T_CtrleAction.xExecute:=TRUE;
	END_IF;
	IF xTmpStopAxis AND T_Visu.T_CtrleAction.xDone AND NOT(T_Visu.T_CtrleAction.xExecute) AND T_Station.THardware.TAxisToolLeft.T_CtrleSingle.xNotMoving AND
	    ((T_Station.THardware.TAxisToolCenter.T_CtrleSingle.xNotMoving AND xMicroRodActive) OR NOT(xMicroRodActive)) AND T_Station.THardware.TAxisToolRight.T_CtrleSingle.xNotMoving AND
	    T_Station.THardware.TAxisToolFeeder.T_CtrleSingle.xNotMoving AND T_Station.THardware.TAxisGrindFeeder.T_CtrleSingle.xNotMoving THEN
		xTmpStopAxis:=FALSE;
	END_IF;

(* Managment Bt Function panel *)
	IF (T_Visu.T_PlcParam.dwActualPage = 10) OR (T_Visu.T_PlcParam.dwActualPage = 110) THEN
		IF NOT(xMicroRodActive) THEN
		(* For MicroWire no Function for move the ToolFeeder to the StartPos-->Cancel Function F5 *)
			wMaskFunctionPanel:=wMaskFunctionPanel AND 16#FFEF;
			T_Visu.ptrT_ExchgParam^.T_BtFunctionPanel.wNotMasktext:=T_Visu.ptrT_ExchgParam^.T_BtFunctionPanel.wNotMasktext OR 16#10;
		END_IF;
	END_IF;
	IF (T_Visu.T_PlcParam.dwActualPage = 20) THEN
		IF NOT(xMicroRodActive) THEN
		(* For MicroWire no Function for move the ToolFeeder to the StartPos-->Cancel Function F5 *)
			wMaskFunctionPanel:=wMaskFunctionPanel AND 16#FFEF;
			T_Visu.ptrT_ExchgParam^.T_BtFunctionPanel.wNotMasktext:=T_Visu.ptrT_ExchgParam^.T_BtFunctionPanel.wNotMasktext OR 16#10;
		END_IF;
	END_IF;
	IF (T_Visu.T_PlcParam.dwActualPage = 310) THEN
		IF NOT(xMicroRodActive) THEN
		(* For MicroWire no Function for no Position to save for ToolFeeder-->Cancel Function F3 and F6 *)
			wMaskFunctionPanel:=wMaskFunctionPanel AND 16#FFDB;
			T_Visu.ptrT_ExchgParam^.T_BtFunctionPanel.wNotMasktext:=T_Visu.ptrT_ExchgParam^.T_BtFunctionPanel.wNotMasktext OR 16#24;
		END_IF;
	END_IF;
	IF (T_Visu.T_PlcParam.dwActualPage = 320) THEN
		IF NOT(xMicroRodActive) THEN
		(* For MicroWire no Function for ToolFeeder-->Cancel Function F1, F2, F3 and F4 *)
			wMaskFunctionPanel:=wMaskFunctionPanel AND 16#0;
			T_Visu.ptrT_ExchgParam^.T_BtFunctionPanel.wNotMasktext:=T_Visu.ptrT_ExchgParam^.T_BtFunctionPanel.wNotMasktext OR 16#FFFF;
		END_IF;
	END_IF;
	RisingEdgeBtFunctionPanel(CLK:=(T_Visu.ptrT_ExchgParam^.T_BtFunctionPanel.wActivBt AND wMaskFunctionPanel) <> 16#0);
	FallingEdgeBtFunctionPanel(CLK:=(T_Visu.ptrT_ExchgParam^.T_BtFunctionPanel.wActivBt AND wMaskFunctionPanel) <> 16#0);
	xTmp:=	NOT(xChangePage)
			AND T_Visu.T_CtrleAction.xDone
			AND NOT(T_Visu.T_CtrleAction.xExecute)
			AND NOT(T_StartUp.T_State.xBlockChangeMovementVisu);
	IF xTmp THEN
		(* Rising edge action *)
		IF RisingEdgeBtFunctionPanel.Q THEN
		(* Init. variable *)
			ii:=1;
			wTmp:=T_Visu.ptrT_ExchgParam^.T_BtFunctionPanel.wActivBt;
			WHILE wTmp <> 16#0 DO
				IF (wTmp AND 16#1) = 16#1 THEN EXIT; END_IF
				wTmp:=ROR(wTmp,1);
				ii:=ii+1;
			END_WHILE
			(* set the new action if present *)
			IF  T_ConfigPage.aiRTrigActionFunctionPanel[ii] <> 0 THEN
				T_Visu.T_CtrleAction.iFunction:= T_ConfigPage.aiRTrigActionFunctionPanel[ii];
				T_Visu.T_CtrleAction.xExecute:=TRUE;
			END_IF
		END_IF
	END_IF

(* Management Bt navigation panel *)
	RisingEdgeTouchScreenNavPanel(CLK:=	T_Visu.ptrT_ExchgParam^.T_TouchScreenNavPanel.wActivBt <> 0);
	FallingEdgeTouchScreenNavPanel(CLK:=T_Visu.ptrT_ExchgParam^.T_TouchScreenNavPanel.wActivBt <> 0);
	xTmp:=	NOT(xChangePage)
			AND T_Visu.T_CtrleAction.xDone
			AND NOT(T_Visu.T_CtrleAction.xExecute)
			AND NOT(T_StartUp.T_State.xBlockChangeMovementVisu)
			AND NOT(T_StartUp.T_State.xBlockVisuNavigation)
			AND ((T_Visu.ptrT_ExchgParam^. T_TouchScreenNavPanel.wNotMasktext AND T_Visu.ptrT_ExchgParam^.T_TouchScreenNavPanel.wActivBt) <> 0);
	IF xTmp THEN
		(* activ action of rising edge *)
		IF RisingEdgeTouchScreenNavPanel.Q THEN
			ii:=1;
			wTmp:=T_Visu.ptrT_ExchgParam^.T_TouchScreenNavPanel.wActivBt;
			WHILE wTmp <> 16#0 DO
				IF (wTmp AND 16#1) = 16#1 THEN EXIT; END_IF
				wTmp:=ROR(wTmp,1);
				ii:=ii+1;
			END_WHILE
			T_Visu.T_CtrleAction.iFunction:=T_ConfigPage.aiFTrigActionTouchScreenNavPanel[ii];
			CASE T_Visu.ptrT_ExchgParam^.T_Visu.bActivSpecialLayer OF
				0: 	wNormalLayerActivTask:=T_Visu.ptrT_ExchgParam^.T_TouchScreenNavPanel.wActivBt;
					wNormalLayerActivPage:=T_Visu.T_CtrleAction.iFunction - 10000;
					T_Visu.ptrT_ExchgParam^.T_TouchScreenNavPanel.wState:=wNormalLayerActivTask;
					wTmpNormalLayerActivTask:=ii;
				1:	wSpecialLayerGeneralActivTask:=T_Visu.ptrT_ExchgParam^.T_TouchScreenNavPanel.wActivBt;
					wSpecialLayerGeneralActivPage:=T_Visu.T_CtrleAction.iFunction - 10000;
					T_Visu.ptrT_ExchgParam^.T_TouchScreenNavPanel.wState:=wSpecialLayerGeneralActivTask;
					wTmpSpecialLayerGeneralActivTask:=ii;
				2:	wSpecialLayerToolRotActivTask:=T_Visu.ptrT_ExchgParam^.T_TouchScreenNavPanel.wActivBt;
					wSpecialLayerToolRotActivPage:=T_Visu.T_CtrleAction.iFunction - 10000;
					T_Visu.ptrT_ExchgParam^.T_TouchScreenNavPanel.wState:=wSpecialLayerToolRotActivTask;
					wTmpSpecialLayerToolRotActivTask:=ii;
				3:	wSpecialLayerWireFeedActivTask:=T_Visu.ptrT_ExchgParam^.T_TouchScreenNavPanel.wActivBt;
					wSpecialLayerWireFeedActivPage:=T_Visu.T_CtrleAction.iFunction - 10000;
					T_Visu.ptrT_ExchgParam^.T_TouchScreenNavPanel.wState:=wSpecialLayerWireFeedActivTask;
					wTmpSpecialLayerWireFeedActivTask:=ii;
				4:	wSpecialLayerGrindAxisActivTask:=T_Visu.ptrT_ExchgParam^.T_TouchScreenNavPanel.wActivBt;
					wSpecialLayerGrindAxisActivPage:=T_Visu.T_CtrleAction.iFunction - 10000;
					T_Visu.ptrT_ExchgParam^.T_TouchScreenNavPanel.wState:=wSpecialLayerGrindAxisActivTask;
					wTmpSpecialLayerGrindAxisActivTask:=ii;
			END_CASE;
			IF ((INT_TO_WORD(T_Visu.ptrT_ExchgParam^.T_TouchScreenBtPanel.iStateBtLeft) AND 16#10) = 16#10) THEN
				T_Visu.T_CtrleAction.iFunction:=3;
				xResetParaListValue:=TRUE;
			END_IF;
			T_Visu.ptrT_ExchgParam^.T_TouchScreenNavPanel.wActivBt:=0;
			T_Visu.T_CtrleAction.xExecute:=TRUE;
		END_IF;
	ELSE
		T_Visu.ptrT_ExchgParam^.T_TouchScreenNavPanel.wActivBt:=0;
	END_IF;
(*22.12.2009: KFS 	{	*)
(* Management BT Tool  (additionel external buttons) only for MicroRod *)
	IF xMicroRodActive THEN
		(* ToolTension button *)
		xTmp:=	NOT(xChangePage) AND T_Visu.T_CtrleAction.xDone AND
				NOT(T_Visu.T_CtrleAction.xExecute) 	AND T_Visu.T_CtrleProcess.xDone AND (bStateMachine <>2);
		IF xTmp THEN
(*03.03.2017: KFS { *)
			RisingEdgeBtToolTension(CLK:=xToolTensionButton);
			IF RisingEdgeBtToolTension.Q THEN
				IF  T_Visu.ptrT_ExchgParam^.T_Cylinder.xToolTension AND	T_Visu.ptrT_ExchgParam^.T_Cylinder.xCylToolLeft AND T_Visu.ptrT_ExchgParam^.T_Cylinder.xCylToolRight	THEN
					T_Visu.T_CtrleAction.iFunction:=510;
					T_Visu.T_CtrleAction.xExecute:=TRUE;
				END_IF;
				IF  NOT (T_Visu.ptrT_ExchgParam^.T_Cylinder.xToolTension) THEN
					T_Visu.T_CtrleAction.iFunction:=510;
					T_Visu.T_CtrleAction.xExecute:=TRUE;
				END_IF;
			END_IF;
			RisingEdgeBtToolLeft(CLK:=xToolLeftButton);
			IF RisingEdgeBtToolLeft.Q THEN
				IF NOT T_Visu.ptrT_ExchgParam^.T_Cylinder.xToolTension  THEN
					T_Visu.T_CtrleAction.iFunction:=511;
					T_Visu.T_CtrleAction.xExecute:=TRUE;
				END_IF;
				IF  T_Visu.ptrT_ExchgParam^.T_Cylinder.xToolTension  AND NOT(T_Visu.ptrT_ExchgParam^.T_Cylinder.xCylToolLeft) THEN
					T_Visu.T_CtrleAction.iFunction:=511;
					T_Visu.T_CtrleAction.xExecute:=TRUE;
				END_IF;
			END_IF;
			RisingEdgeBtToolRight(CLK:=xToolRightButton);
			IF RisingEdgeBtToolRight.Q THEN
				IF NOT T_Visu.ptrT_ExchgParam^.T_Cylinder.xToolTension  THEN
					T_Visu.T_CtrleAction.iFunction:=512;
					T_Visu.T_CtrleAction.xExecute:=TRUE;
				END_IF;
				IF  T_Visu.ptrT_ExchgParam^.T_Cylinder.xToolTension  AND NOT(T_Visu.ptrT_ExchgParam^.T_Cylinder.xCylToolRight) THEN
					T_Visu.T_CtrleAction.iFunction:=512;
					T_Visu.T_CtrleAction.xExecute:=TRUE;
				END_IF;
			END_IF;
(*03.03.2017: KFS } *)
			RisingEdgeBtToolCenter(CLK:=xToolCenterButton);
			IF RisingEdgeBtToolCenter.Q THEN
				T_Visu.T_CtrleAction.iFunction:=513;
				T_Visu.T_CtrleAction.xExecute:=TRUE;
			END_IF;
			RisingEdgeBtToolPrismaLeft(CLK:=xToolPrismaLeftButton);
			IF RisingEdgeBtToolPrismaLeft.Q THEN
				T_Visu.T_CtrleAction.iFunction:=514;
				T_Visu.T_CtrleAction.xExecute:=TRUE;
			END_IF;
			RisingEdgeBtToolPrismaRight(CLK:=xToolPrismaRightButton);
			IF RisingEdgeBtToolPrismaRight.Q THEN
				T_Visu.T_CtrleAction.iFunction:=515;
				T_Visu.T_CtrleAction.xExecute:=TRUE;
			END_IF;
		ELSE
			IF   NOT(T_Visu.T_CtrleAction.xExecute) AND T_Visu.T_CtrleAction.xDone  THEN
				RisingEdgeBtToolTension(CLK:=FALSE);
				RisingEdgeBtToolLeft(CLK:=FALSE);
				RisingEdgeBtToolRight(CLK:=FALSE);
				RisingEdgeBtToolCenter(CLK:=FALSE);
				RisingEdgeBtToolPrismaLeft(CLK:=FALSE);
				RisingEdgeBtToolPrismaRight(CLK:=FALSE);
			END_IF;
		END_IF;
	END_IF;
(*22.12.2009: KFS 	}	*)
(************************************************************************************************************************************************************************)
(*********end of the managment of the external start-stop button, special button and function button and task button and external tool buttons********)
(************************************************************************************************************************************************************************)

(* set system level *)
	IF (T_Visu.ptrT_ExchgParam^.T_Visu.T_Level.iPwSystem <> 999) AND (T_Visu.T_PlcParam.dwActualPage = 40) THEN
		IF T_Visu.ptrT_ExchgParam^.T_Visu.T_Level.iPwSystem = iPwSystem THEN
		(* pw correct *)
			T_Visu.ptrT_ExchgParam^.T_Visu.T_Level.iActLevel:=2;
			T_Visu.ptrT_ExchgParam^.T_Visu.T_Message.iState:=2;
		(* wrong pw *)
		ELSE 	T_Visu.ptrT_ExchgParam^.T_Visu.T_Message.iState:=3; END_IF
		T_Visu.ptrT_ExchgParam^.T_Visu.T_Level.iPwSystem:=999;
	END_IF
	IF (T_Visu.T_PlcParam.dwActualPage = 40) THEN
		RisingEdgeDynPassword(CLK:=TRUE);
		IF RisingEdgeDynPassword.Q THEN
			fbGetCpuAccount;
			fbPwSystem(	dwCounter:=fbGetCpuAccount.fbGetCpuCounter.dwCpuCntHi+fbGetCpuAccount.fbGetCpuCounter.dwCpuCntLo,
						iRandom=>T_Visu.ptrT_ExchgParam^.T_Visu.T_Level.iRandom,
						iPwSystem=>iPwSystem);
		END_IF;
	ELSE
		RisingEdgeDynPassword(CLK:=FALSE);
	END_IF;

(************************************************************************************************************************************************************************)
(**********************************						Profile Management Start						****************************************)
(************************************************************************************************************************************************************************)

(* Update profile list *)
	IF xUpdateProfileList THEN
		xTmp:= 	iPointerListProfile > 0
				AND (iPointerListProfile+4) <= csiMaxProfile;
		IF xTmp THEN
			jj:=1;
			FOR ii:=iPointerListProfile TO iPointerListProfile+4 DO
				T_Visu.ptrT_ExchgParam^.T_ProfileCommon.T_ProfileList[jj].iNumber:=ii;
				T_Visu.ptrT_ExchgParam^.T_ProfileCommon.T_ProfileList[jj].sName:=T_NovRam.T_Data.T_IDProfileStation[ii].sName;
				jj:=jj+1;
			END_FOR
		END_IF
		(* confirm update *)
		xUpdateProfileList:=FALSE;
	END_IF

(* Compare Profile and Process value *)
	xTmp:=	(T_Visu.ptrT_ExchgParam^.T_StationCommon.T_InfoProcess.iProfile <> 0);
	IF xTmp THEN
		fbCompareProfileProcessValue(T_Data_ProcessImageLoadData:=T_NovRam.T_Data.T_ProcessImageLoadData,
									T_Data_ProcessImageData:=T_NovRam.T_Data.T_ProcessImageData,
									xMicroRodActive:=xMicroRodActive);
		T_Visu.ptrT_ExchgParam^.T_StationCommon.T_InfoProcess.xOnlineValueModified:=fbCompareProfileProcessValue.xProcessValueModified;
	END_IF

(* monitor change actual profile common *)
	IF (T_Visu.T_PlcParam.dwActualPage = 130) THEN
		IF T_Visu.ptrT_ExchgParam^.T_ProfileCommon.T_Id.iNumber<>iActualActiveProfile THEN
			IF T_Visu.T_CtrleAction.xDone THEN
				(* set value from selected profile *)
				T_Visu.ptrT_ExchgParam^.T_ProfileCommon.T_Id.sName
					:=T_NovRam.T_Data.T_IDProfileStation[T_Visu.ptrT_ExchgParam^.T_ProfileCommon.T_Id.iNumber].sName;
				(* save value from selected profile *)
				iActualActiveProfile:=T_Visu.ptrT_ExchgParam^.T_ProfileCommon.T_Id.iNumber;
			END_IF
		END_IF
	END_IF

(* Pointer Profile List Up/Down Slow *)
	RisingEdgePtrProfileListUpDown(CLK:=	T_Visu.ptrT_ExchgParam^.T_ProfileCommon.T_ProfileManage.xListProfileUp
										OR T_Visu.ptrT_ExchgParam^.T_ProfileCommon.T_ProfileManage.xListProfileDown);
	IF RisingEdgePtrProfileListUpDown.Q THEN
		IF T_Visu.ptrT_ExchgParam^.T_ProfileCommon.T_ProfileManage.xListProfileUp THEN
			iPointerListProfile:=iPointerListProfile-5;
		ELSE iPointerListProfile:=iPointerListProfile+5; END_IF
		(* min/max=1/6 *)
		IF iPointerListProfile>(csiMaxProfile -5) THEN iPointerListProfile:=(csiMaxProfile - 4); END_IF
		IF iPointerListProfile<0 THEN iPointerListProfile:=1; END_IF
		T_Visu.ptrT_ExchgParam^.T_ProfileCommon.T_ProfileManage.xListProfileUp:=FALSE;
		T_Visu.ptrT_ExchgParam^.T_ProfileCommon.T_ProfileManage.xListProfileDown:=FALSE;
		(* Update display  list *)
		xUpdateProfileList:=TRUE;
	END_IF

(* Pointer Profile List Up/Down Fast *)
	RisingEdgePtrProfileListUpDown(CLK:=	T_Visu.ptrT_ExchgParam^.T_ProfileCommon.T_ProfileManage.xListProfileUpFast
										OR T_Visu.ptrT_ExchgParam^.T_ProfileCommon.T_ProfileManage.xListProfileDownFast);
	IF RisingEdgePtrProfileListUpDown.Q THEN
		IF T_Visu.ptrT_ExchgParam^.T_ProfileCommon.T_ProfileManage.xListProfileUpFast THEN
			iPointerListProfile:=iPointerListProfile-10;
		ELSE iPointerListProfile:=iPointerListProfile+10; END_IF
		(* min/max=1/6 *)
		IF iPointerListProfile>(csiMaxProfile -5) THEN iPointerListProfile:=(csiMaxProfile - 4); END_IF
		IF iPointerListProfile<0 THEN iPointerListProfile:=1; END_IF
		T_Visu.ptrT_ExchgParam^.T_ProfileCommon.T_ProfileManage.xListProfileUpFast:=FALSE;
		T_Visu.ptrT_ExchgParam^.T_ProfileCommon.T_ProfileManage.xListProfileDownFast:=FALSE;
		(* Update display  list *)
		xUpdateProfileList:=TRUE;
	END_IF

(************************************************************************************************************************************************************************)
(**********************************						Profile Management End						****************************************)
(************************************************************************************************************************************************************************)

(* Display info or warning message *)
	RisingEdgeKeySwitch1(CLK:=xSecurityKey);
	FailingEdgeKeySwitch1(CLK:=xSecurityKey);
	IF T_Visu.ptrT_ExchgParam^.T_Visu.T_Message.iState <> 0 THEN
		(* info message *)
		IF T_Visu.ptrT_ExchgParam^.T_Visu.T_Message.iState < 100THEN
		(* activ message during 3s, after that the message will be cleared *)
			TimerDisplayMessage(IN:=TRUE,PT:=T#3s);
			IF TimerDisplayMessage.Q THEN
				T_Visu.ptrT_ExchgParam^.T_Visu.T_Message.iState:=0;
				TimerDisplayMessage(IN:=FALSE);
			END_IF
			IF (T_Visu.ptrT_ExchgParam^.T_Visu.T_Message.iState = 2) THEN
				IF (TimerDisplayMessage.ET > T#0.5s) THEN
					T_Visu.ptrT_ExchgParam^.T_Visu.T_Message.iState:=0;
					TimerDisplayMessage(IN:=FALSE);
				END_IF;
			END_IF;
		(* disable timer *)
		ELSE TimerDisplayMessage(IN:=FALSE); END_IF

		(* warning message *)
		xTmp:=	(T_Visu.ptrT_ExchgParam^.T_Visu.T_Message.iState > 100 AND T_Visu.ptrT_ExchgParam^.T_Visu.T_Message.iState <200)
				AND T_Visu.T_CtrleAction.xDone;
		RisingEdgeReleaseWarning(CLK:=wActivBtLeft <> 16#0 OR T_Visu.ptrT_ExchgParam^.T_BtFunctionPanel.wActivBt <> 16#0);
		(* the warning will be cleared by the operator *)
		IF xTmp AND (RisingEdgeReleaseWarning.Q OR RisingEdgeKeySwitch1.Q OR FailingEdgeKeySwitch1.Q) THEN
			IF (T_Visu.ptrT_ExchgParam^.T_Visu.T_Message.iState <> 120) THEN
				T_Visu.ptrT_ExchgParam^.T_Visu.T_Message.iState:=0;
			END_IF;
		END_IF
	END_IF

(* Monitor dynamic error text *)
	xTmp:=	T_Visu.ptrT_ExchgParam^.T_Visu.T_Message.sDynamicTextEnglish <> ''
			AND T_Visu.ptrT_ExchgParam^.T_Visu.T_Message.iState <> 401;
	IF xTmp THEN
		bStateMachine:=0;
		T_Visu.ptrT_ExchgParam^.T_Visu.T_Message.iState:=401;
		xSetStateMachine:=TRUE;
		xCheckQuitError:=TRUE;
	END_IF
	IF xCheckQuitError THEN
		IF (T_Visu.ptrT_ExchgParam^.T_Visu.T_Message.iState <> 401) THEN
			xSetStateMachine:=TRUE;
			xCheckQuitError:=FALSE;
			IF NOT(T_TwinSafeOut.QxContactor_K3) OR NOT(T_TwinSafeOut.QxContactor_K4) THEN
				bStateMachine:=3;
			ELSE
				bStateMachine:=1;
			END_IF;
		END_IF;
	END_IF;
	IF NOT(T_TwinSafeIn.IxPowerSupplyEcoStep) THEN
		bStateMachine:=4;
	END_IF;
	IF xSetStateMachine THEN
		xSetStateMachine:=FALSE;
		T_Visu.ptrT_ExchgParam^.T_SafetyCtrl.bStateAutoGeometry:=bStateMachine;
		T_Visu.ptrT_ExchgParam^.T_SafetyCtrl.bStateAutoGroove:=bStateMachine;
		T_Visu.ptrT_ExchgParam^.T_SafetyCtrl.bStateReference:=bStateMachine;
		T_Visu.ptrT_ExchgParam^.T_SafetyCtrl.bStateToolCalibration:=bStateMachine;
		T_Visu.ptrT_ExchgParam^.T_SafetyCtrl.bStateToolTorque:=bStateMachine;
		T_Visu.ptrT_ExchgParam^.T_SafetyCtrl.bStateTeachInToolLeft:=bStateMachine;
		T_Visu.ptrT_ExchgParam^.T_SafetyCtrl.bStateTeachInToolCenter:=bStateMachine;
		T_Visu.ptrT_ExchgParam^.T_SafetyCtrl.bStateTeachInToolRight:=bStateMachine;
		T_Visu.ptrT_ExchgParam^.T_SafetyCtrl.bStateTeachInToolFeeder:=bStateMachine;
		T_Visu.ptrT_ExchgParam^.T_SafetyCtrl.bStateReferenceMaxToolLength:=bStateMachine;
		T_Visu.ptrT_ExchgParam^.T_SafetyCtrl.bStateTeachInGrindFeeder:=bStateMachine;
		T_Visu.ptrT_ExchgParam^.T_StationCommon.iWireFeederRefIndexState:=BYTE_TO_INT(bStateMachine);
	END_IF;

(* Reset settled value on the parameter list, without saved *)
	IF xResetParaListValue OR T_Visu.T_CtrleAction.xResetParaListValue THEN
		T_Visu.T_CtrleAction.xResetParaListValue:=FALSE;
		xResetParaListValue:=FALSE;
		T_Visu.ptrT_ExchgParam^.T_TeachIn.TParam_ToolLeft:=T_NovRAM.T_Data.T_Standard.T_TeachINToolLeft;
		T_Visu.ptrT_ExchgParam^.T_TeachIn.TParam_ToolCenter:=T_NovRAM.T_Data.T_Standard.T_TeachINToolCenter;
		T_Visu.ptrT_ExchgParam^.T_TeachIn.TParam_ToolRight:=T_NovRAM.T_Data.T_Standard.T_TeachINToolRight;
		T_Visu.ptrT_ExchgParam^.T_TeachIn.TParam_ToolFeeder:=T_NovRAM.T_Data.T_Standard.T_TeachINToolFeeder;
		T_Visu.ptrT_ExchgParam^.T_TeachIn.TParam_GrindFeeder:=T_NovRAM.T_Data.T_Standard.T_TeachINGrindFeeder;
		T_Visu.ptrT_ExchgParam^.T_TeachIn.TParam_AxisPosition:=T_NovRAM.T_Data.T_Standard.T_AxisPosition;
		T_Visu.ptrT_ExchgParam^.T_StationCommon.iConfigMachineType:=T_NovRAM.T_Data.T_Standard.T_MachineConfig.iConfigMachineType;
		T_Visu.ptrT_ExchgParam^.T_StationCommon.iConfigAxisType:=T_NovRAM.T_Data.T_Standard.T_MachineConfig.iConfigAxisType;
		T_Visu.ptrT_ExchgParam^.T_StationCommon.iConfigVisuNavigation:=T_NovRAM.T_Data.T_Standard.T_MachineConfig.iConfigVisuNavigation;
		T_Visu.ptrT_ExchgParam^.T_StationCommon.rConfigMaxToolLength:=T_NovRAM.T_Data.T_Standard.T_MachineConfig.rConfigMaxToolLength;
		T_Visu.ptrT_ExchgParam^.T_StationCommon.T_ParamToolTensionSystem:=T_NovRAM.T_Data.T_Standard.T_ToolTensionSystem;
		T_Visu.ptrT_ExchgParam^.T_Cylinder.T_ParamToolTension:=T_NovRAM.T_Data.T_Standard.T_Cyl_ToolTension;
		T_Visu.ptrT_ExchgParam^.T_StationCommon.T_AutoGeometryPara:=T_NovRAM.T_Data.T_ProcessImageData.T_AutoGeometryPara;
		T_Visu.ptrT_ExchgParam^.T_StationCommon.T_AutoGroovePara:=T_NovRAM.T_Data.T_ProcessImageData.T_AutoGroovePara;
		T_Visu.ptrT_ExchgParam^.T_StationCommon.T_CalibrationPara:=T_NovRAM.T_Data.T_ProcessImageData.T_CalibrationPara;
		T_Visu.ptrT_ExchgParam^.T_StationCommon.T_ProcessPara:=T_NovRAM.T_Data.T_ProcessImageData.T_ProcessPara;
		T_Visu.ptrT_ExchgParam^.T_StationCommon.T_InfoProcess.iProfile:=T_Visu.ptrT_ExchgParam^.T_ProfileCommon.T_Id.iNumber;
		T_Visu.ptrT_ExchgParam^.T_StationCommon.T_InfoProcess.sProfileName:=T_NovRam.T_Data.T_IDProfileStation[T_Visu.ptrT_ExchgParam^.T_ProfileCommon.T_Id.iNumber].sName;
		T_Visu.ptrT_ExchgParam^.T_GeometryCommon.T_Geometry:=T_NovRAM.T_Data.T_ProcessImageData.T_GeometryPara;
		T_Visu.ptrT_ExchgParam^.T_StationCommon.T_PrismPara:=T_NovRAM.T_Data.T_ProcessImageData.T_PrismPara;
		T_Visu.ptrT_ExchgParam^.T_GeometryCommon.rMinToolDiameter:=T_NovRAM.T_Data.T_ProcessImageData.T_PrismPara.rToolDiameterMin;
		T_Visu.ptrT_ExchgParam^.T_GeometryCommon.rMaxToolDiameter:=T_NovRAM.T_Data.T_ProcessImageData.T_PrismPara.rToolDiameterMax;
		T_Visu.ptrT_ExchgParam^.T_GeometryCommon.rMinToolLength:=0.1;
		T_Visu.ptrT_ExchgParam^.T_GeometryCommon.rMaxToolLength:=T_NovRAM.T_Data.T_Standard.T_MachineConfig.rConfigMaxToolLength;
		T_Visu.ptrT_ExchgParam^.T_StationCommon.rConfigMaxToolLengthOriginal:=T_NovRAM.T_Data.T_Standard.T_MachineConfig.rConfigMaxToolLengthOriginal;
	END_IF;

(* Monitoring Process value *)
	IF T_Process.xReferenced THEN T_Visu.ptrT_ExchgParam^.T_Machine.T_Process.wState:=T_Visu.ptrT_ExchgParam^.T_Machine.T_Process.wState OR 16#1;
		ELSE T_Visu.ptrT_ExchgParam^.T_Machine.T_Process.wState:=T_Visu.ptrT_ExchgParam^.T_Machine.T_Process.wState AND 16#FE; END_IF
	IF NOT(T_Process.xEnd) THEN T_Visu.ptrT_ExchgParam^.T_Machine.T_Process.wState:=T_Visu.ptrT_ExchgParam^.T_Machine.T_Process.wState OR 16#2;
		ELSE T_Visu.ptrT_ExchgParam^.T_Machine.T_Process.wState:=T_Visu.ptrT_ExchgParam^.T_Machine.T_Process.wState AND 16#FD; END_IF
	IF T_Process.xError THEN T_Visu.ptrT_ExchgParam^.T_Machine.T_Process.wState:=T_Visu.ptrT_ExchgParam^.T_Machine.T_Process.wState OR 16#4;
		ELSE T_Visu.ptrT_ExchgParam^.T_Machine.T_Process.wState:=T_Visu.ptrT_ExchgParam^.T_Machine.T_Process.wState AND 16#FB; END_IF
	IF T_Process.xRdy THEN T_Visu.ptrT_ExchgParam^.T_Machine.T_Process.wState:=T_Visu.ptrT_ExchgParam^.T_Machine.T_Process.wState OR 16#8;
		ELSE T_Visu.ptrT_ExchgParam^.T_Machine.T_Process.wState:=T_Visu.ptrT_ExchgParam^.T_Machine.T_Process.wState AND 16#F7; END_IF
	IF T_Process.xEnd THEN T_Visu.ptrT_ExchgParam^.T_Machine.T_Process.wState:=T_Visu.ptrT_ExchgParam^.T_Machine.T_Process.wState OR 16#10;
		ELSE T_Visu.ptrT_ExchgParam^.T_Machine.T_Process.wState:=T_Visu.ptrT_ExchgParam^.T_Machine.T_Process.wState AND 16#EF; END_IF
	IF T_Process.xProcessHold THEN T_Visu.ptrT_ExchgParam^.T_Machine.T_Process.wState:=T_Visu.ptrT_ExchgParam^.T_Machine.T_Process.wState OR 16#40;
		ELSE T_Visu.ptrT_ExchgParam^.T_Machine.T_Process.wState:=T_Visu.ptrT_ExchgParam^.T_Machine.T_Process.wState AND 16#BF; END_IF
	IF T_Process.xStop THEN T_Visu.ptrT_ExchgParam^.T_Machine.T_Process.wState:=T_Visu.ptrT_ExchgParam^.T_Machine.T_Process.wState OR 16#80;
		ELSE T_Visu.ptrT_ExchgParam^.T_Machine.T_Process.wState:=T_Visu.ptrT_ExchgParam^.T_Machine.T_Process.wState AND 16#7F; END_IF

(* Monitoring Station value *)
	IF T_Station.TControl.xEnd AND T_Station.TControl.xRdy AND T_Station.TControl.xEnable THEN
		T_Visu.ptrT_ExchgParam^.T_StationCommon.bStateMachine:=T_Visu.ptrT_ExchgParam^.T_StationCommon.bStateMachine OR 16#1;
	ELSE
		T_Visu.ptrT_ExchgParam^.T_StationCommon.bStateMachine:=T_Visu.ptrT_ExchgParam^.T_StationCommon.bStateMachine AND 16#FE;
	END_IF;
	IF NOT(T_Station.TControl.xEnd) AND T_Station.TControl.xRdy AND T_Station.TControl.xEnable THEN
		T_Visu.ptrT_ExchgParam^.T_StationCommon.bStateMachine:=T_Visu.ptrT_ExchgParam^.T_StationCommon.bStateMachine OR 16#2;
	ELSE
		T_Visu.ptrT_ExchgParam^.T_StationCommon.bStateMachine:=T_Visu.ptrT_ExchgParam^.T_StationCommon.bStateMachine AND 16#FD;
	END_IF;
	IF T_Station.TControl.xError THEN
		T_Visu.ptrT_ExchgParam^.T_StationCommon.bStateMachine:=T_Visu.ptrT_ExchgParam^.T_StationCommon.bStateMachine OR 16#4;
	ELSE
		T_Visu.ptrT_ExchgParam^.T_StationCommon.bStateMachine:=T_Visu.ptrT_ExchgParam^.T_StationCommon.bStateMachine AND 16#FB;
	END_IF;
	IF T_Station.TControl.xReferenced THEN
		T_Visu.ptrT_ExchgParam^.T_StationCommon.bStateMachine:=T_Visu.ptrT_ExchgParam^.T_StationCommon.bStateMachine OR 16#8;
	ELSE
		T_Visu.ptrT_ExchgParam^.T_StationCommon.bStateMachine:=T_Visu.ptrT_ExchgParam^.T_StationCommon.bStateMachine AND 16#F7;
	END_IF;

(* Monitoring for the visu of the state of the machine *)
	T_Visu.ptrT_ExchgParam^.T_StationCommon.bStateMachineLED:=16#0;
	IF T_Station.TControl.xError OR T_Station.THardware.TAxisToolLeft.T_CtrleSingle.xErr OR (T_Station.THardware.TAxisToolCenter.T_CtrleSingle.xErr AND xMicroRodActive) OR
	    T_Station.THardware.TAxisToolRight.T_CtrleSingle.xErr OR T_Station.THardware.TAxisToolFeeder.T_CtrleSingle.xErr OR T_Station.THardware.TAxisGrindFeeder.T_CtrleSingle.xErr OR
	     (T_ExchgParam.T_Visu.T_Message.iState = 401) THEN
		T_Visu.ptrT_ExchgParam^.T_StationCommon.bStateMachineLED:=16#4;
	ELSIF NOT(T_Station.TControl.xEnd) OR NOT(T_Process.xEnd) OR T_Station.TControl.xActiveMovement THEN
		T_Visu.ptrT_ExchgParam^.T_StationCommon.bStateMachineLED:=16#2;
	ELSE
		T_Visu.ptrT_ExchgParam^.T_StationCommon.bStateMachineLED:=16#1;
	END_IF;
	IF (T_Visu.ptrT_ExchgParam^.T_StationCommon.bStateMachineLED <> 16#4) THEN
		IF NOT(T_TwinSafeOut.QxContactor_K3) OR NOT(T_TwinSafeOut.QxContactor_K4) THEN
			T_Visu.ptrT_ExchgParam^.T_StationCommon.bStateMachineLED:=16#0;
		END_IF;
	END_IF

(* Monitoring Axis value *)
	(* ToolLeft Monitoring *)
	IF T_Station.THardware.TAxisToolLeft.T_CtrleSingle.xPower THEN
		T_Visu.ptrT_ExchgParam^.T_StationCommon.bStateAxisReelLeft:=T_Visu.ptrT_ExchgParam^.T_StationCommon.bStateAxisReelLeft OR 16#1;
	ELSE
		T_Visu.ptrT_ExchgParam^.T_StationCommon.bStateAxisReelLeft:=T_Visu.ptrT_ExchgParam^.T_StationCommon.bStateAxisReelLeft AND 16#FE;
	END_IF;
	IF NOT(T_Station.THardware.TAxisToolLeft.T_CtrleSingle.xNotMoving) THEN
		T_Visu.ptrT_ExchgParam^.T_StationCommon.bStateAxisReelLeft:=T_Visu.ptrT_ExchgParam^.T_StationCommon.bStateAxisReelLeft OR 16#2;
	ELSE
		T_Visu.ptrT_ExchgParam^.T_StationCommon.bStateAxisReelLeft:=T_Visu.ptrT_ExchgParam^.T_StationCommon.bStateAxisReelLeft AND 16#FD;
	END_IF;
	IF T_Station.THardware.TAxisToolLeft.T_CtrleSingle.xErr THEN
		T_Visu.ptrT_ExchgParam^.T_StationCommon.bStateAxisReelLeft:=T_Visu.ptrT_ExchgParam^.T_StationCommon.bStateAxisReelLeft OR 16#4;
	ELSE
		T_Visu.ptrT_ExchgParam^.T_StationCommon.bStateAxisReelLeft:=T_Visu.ptrT_ExchgParam^.T_StationCommon.bStateAxisReelLeft AND 16#FB;
	END_IF;
	(* ToolRight Monitoring *)
	IF T_Station.THardware.TAxisToolRight.T_CtrleSingle.xPower THEN
		T_Visu.ptrT_ExchgParam^.T_StationCommon.bStateAxisReelRight:=T_Visu.ptrT_ExchgParam^.T_StationCommon.bStateAxisReelRight OR 16#1;
	ELSE
		T_Visu.ptrT_ExchgParam^.T_StationCommon.bStateAxisReelRight:=T_Visu.ptrT_ExchgParam^.T_StationCommon.bStateAxisReelRight AND 16#FE;
	END_IF;
	IF NOT(T_Station.THardware.TAxisToolRight.T_CtrleSingle.xNotMoving) THEN
		T_Visu.ptrT_ExchgParam^.T_StationCommon.bStateAxisReelRight:=T_Visu.ptrT_ExchgParam^.T_StationCommon.bStateAxisReelRight OR 16#2;
	ELSE
		T_Visu.ptrT_ExchgParam^.T_StationCommon.bStateAxisReelRight:=T_Visu.ptrT_ExchgParam^.T_StationCommon.bStateAxisReelRight AND 16#FD;
	END_IF;
	IF T_Station.THardware.TAxisToolRight.T_CtrleSingle.xErr THEN
		T_Visu.ptrT_ExchgParam^.T_StationCommon.bStateAxisReelRight:=T_Visu.ptrT_ExchgParam^.T_StationCommon.bStateAxisReelRight OR 16#4;
	ELSE
		T_Visu.ptrT_ExchgParam^.T_StationCommon.bStateAxisReelRight:=T_Visu.ptrT_ExchgParam^.T_StationCommon.bStateAxisReelRight AND 16#FB;
	END_IF;
	IF T_Station.THardware.TAxisToolRight.T_CtrleSingle.xSlave THEN
		T_Visu.ptrT_ExchgParam^.T_StationCommon.bStateAxisReelRight:=T_Visu.ptrT_ExchgParam^.T_StationCommon.bStateAxisReelRight OR 16#8;
	ELSE
		T_Visu.ptrT_ExchgParam^.T_StationCommon.bStateAxisReelRight:=T_Visu.ptrT_ExchgParam^.T_StationCommon.bStateAxisReelRight AND 16#F7;
	END_IF;
	(* ToolCenter Monitoring *)
	IF T_Station.THardware.TAxisToolCenter.T_CtrleSingle.xPower THEN
		T_Visu.ptrT_ExchgParam^.T_StationCommon.bStateAxisReelCenter:=T_Visu.ptrT_ExchgParam^.T_StationCommon.bStateAxisReelCenter OR 16#1;
	ELSE
		T_Visu.ptrT_ExchgParam^.T_StationCommon.bStateAxisReelCenter:=T_Visu.ptrT_ExchgParam^.T_StationCommon.bStateAxisReelCenter AND 16#FE;
	END_IF;
	IF NOT(T_Station.THardware.TAxisToolCenter.T_CtrleSingle.xNotMoving) THEN
		T_Visu.ptrT_ExchgParam^.T_StationCommon.bStateAxisReelCenter:=T_Visu.ptrT_ExchgParam^.T_StationCommon.bStateAxisReelCenter OR 16#2;
	ELSE
		T_Visu.ptrT_ExchgParam^.T_StationCommon.bStateAxisReelCenter:=T_Visu.ptrT_ExchgParam^.T_StationCommon.bStateAxisReelCenter AND 16#FD;
	END_IF;
	IF T_Station.THardware.TAxisToolCenter.T_CtrleSingle.xErr THEN
		T_Visu.ptrT_ExchgParam^.T_StationCommon.bStateAxisReelCenter:=T_Visu.ptrT_ExchgParam^.T_StationCommon.bStateAxisReelCenter OR 16#4;
	ELSE
		T_Visu.ptrT_ExchgParam^.T_StationCommon.bStateAxisReelCenter:=T_Visu.ptrT_ExchgParam^.T_StationCommon.bStateAxisReelCenter AND 16#FB;
	END_IF;
	IF T_Station.THardware.TAxisToolCenter.T_CtrleSingle.xSlave THEN
		T_Visu.ptrT_ExchgParam^.T_StationCommon.bStateAxisReelCenter:=T_Visu.ptrT_ExchgParam^.T_StationCommon.bStateAxisReelCenter OR 16#8;
	ELSE
		T_Visu.ptrT_ExchgParam^.T_StationCommon.bStateAxisReelCenter:=T_Visu.ptrT_ExchgParam^.T_StationCommon.bStateAxisReelCenter AND 16#F7;
	END_IF;
	(* ToolFeeder Monitoring *)
	IF T_Station.THardware.TAxisToolFeeder.T_CtrleSingle.xPower THEN
		T_Visu.ptrT_ExchgParam^.T_StationCommon.bStateAxisWireFeeder:=T_Visu.ptrT_ExchgParam^.T_StationCommon.bStateAxisWireFeeder OR 16#1;
	ELSE
		T_Visu.ptrT_ExchgParam^.T_StationCommon.bStateAxisWireFeeder:=T_Visu.ptrT_ExchgParam^.T_StationCommon.bStateAxisWireFeeder AND 16#FE;
	END_IF;
	IF NOT(T_Station.THardware.TAxisToolFeeder.T_CtrleSingle.xNotMoving) THEN
		T_Visu.ptrT_ExchgParam^.T_StationCommon.bStateAxisWireFeeder:=T_Visu.ptrT_ExchgParam^.T_StationCommon.bStateAxisWireFeeder OR 16#2;
	ELSE
		T_Visu.ptrT_ExchgParam^.T_StationCommon.bStateAxisWireFeeder:=T_Visu.ptrT_ExchgParam^.T_StationCommon.bStateAxisWireFeeder AND 16#FD;
	END_IF;
	IF T_Station.THardware.TAxisToolFeeder.T_CtrleSingle.xErr THEN
		T_Visu.ptrT_ExchgParam^.T_StationCommon.bStateAxisWireFeeder:=T_Visu.ptrT_ExchgParam^.T_StationCommon.bStateAxisWireFeeder OR 16#4;
	ELSE
		T_Visu.ptrT_ExchgParam^.T_StationCommon.bStateAxisWireFeeder:=T_Visu.ptrT_ExchgParam^.T_StationCommon.bStateAxisWireFeeder AND 16#FB;
	END_IF;
	IF T_Station.THardware.TAxisToolFeeder.T_CtrleSingle.xSlave THEN
		T_Visu.ptrT_ExchgParam^.T_StationCommon.bStateAxisWireFeeder:=T_Visu.ptrT_ExchgParam^.T_StationCommon.bStateAxisWireFeeder OR 16#8;
	ELSE
		T_Visu.ptrT_ExchgParam^.T_StationCommon.bStateAxisWireFeeder:=T_Visu.ptrT_ExchgParam^.T_StationCommon.bStateAxisWireFeeder AND 16#F7;
	END_IF;
	(* GrindFeeder Monitoring *)
	IF T_Station.THardware.TAxisGrindFeeder.T_CtrleSingle.xPower THEN
		T_Visu.ptrT_ExchgParam^.T_StationCommon.bStateAxisGrind:=T_Visu.ptrT_ExchgParam^.T_StationCommon.bStateAxisGrind OR 16#1;
	ELSE
		T_Visu.ptrT_ExchgParam^.T_StationCommon.bStateAxisGrind:=T_Visu.ptrT_ExchgParam^.T_StationCommon.bStateAxisGrind AND 16#FE;
	END_IF;
	IF NOT(T_Station.THardware.TAxisGrindFeeder.T_CtrleSingle.xNotMoving) THEN
		T_Visu.ptrT_ExchgParam^.T_StationCommon.bStateAxisGrind:=T_Visu.ptrT_ExchgParam^.T_StationCommon.bStateAxisGrind OR 16#2;
	ELSE
		T_Visu.ptrT_ExchgParam^.T_StationCommon.bStateAxisGrind:=T_Visu.ptrT_ExchgParam^.T_StationCommon.bStateAxisGrind AND 16#FD;
	END_IF;
	IF T_Station.THardware.TAxisGrindFeeder.T_CtrleSingle.xErr THEN
		T_Visu.ptrT_ExchgParam^.T_StationCommon.bStateAxisGrind:=T_Visu.ptrT_ExchgParam^.T_StationCommon.bStateAxisGrind OR 16#4;
	ELSE
		T_Visu.ptrT_ExchgParam^.T_StationCommon.bStateAxisGrind:=T_Visu.ptrT_ExchgParam^.T_StationCommon.bStateAxisGrind AND 16#FB;
	END_IF;
	IF T_Station.THardware.TAxisGrindFeeder.T_CtrleSingle.xSlave THEN
		T_Visu.ptrT_ExchgParam^.T_StationCommon.bStateAxisGrind:=T_Visu.ptrT_ExchgParam^.T_StationCommon.bStateAxisGrind OR 16#8;
	ELSE
		T_Visu.ptrT_ExchgParam^.T_StationCommon.bStateAxisGrind:=T_Visu.ptrT_ExchgParam^.T_StationCommon.bStateAxisGrind AND 16#F7;
	END_IF;
	(* General Actual Axis value *)
	T_Visu.ptrT_ExchgParam^.T_InfoValueCommon.rActualToolRotSpeed:=T_Station.THardware.TAxisToolLeft.T_LiveValue.lrActualVelocity;
	IF (T_Visu.ptrT_ExchgParam^.T_TeachIn.iSelectAxisToolRotation = 1) THEN
		T_Visu.ptrT_ExchgParam^.T_StationCommon.rActualToolRotationSpeed:=T_Station.THardware.TAxisToolLeft.T_LiveValue.lrActualVelocity;
	END_IF;
	IF (T_Visu.ptrT_ExchgParam^.T_TeachIn.iSelectAxisToolRotation = 2) THEN
		T_Visu.ptrT_ExchgParam^.T_StationCommon.rActualToolRotationSpeed:=T_Station.THardware.TAxisToolCenter.T_LiveValue.lrActualVelocity;
	END_IF;
	IF (T_Visu.ptrT_ExchgParam^.T_TeachIn.iSelectAxisToolRotation = 3) THEN
		T_Visu.ptrT_ExchgParam^.T_StationCommon.rActualToolRotationSpeed:=T_Station.THardware.TAxisToolRight.T_LiveValue.lrActualVelocity;
	END_IF;
	IF xMicroRodActive THEN
		IF (T_Visu.T_PlcParam.dwActualPage = 10) OR (T_Visu.T_PlcParam.dwActualPage = 20) THEN
			T_Visu.ptrT_ExchgParam^.T_InfoValueCommon.rActualWireFeedPosition:=	T_Station.THardware.TAxisToolFeeder.T_LiveValue.lrActualPosition -
																						T_NovRam.T_Data.T_ProcessImageData.T_ProcessPara.rStartPosToolFeedAuto;
		END_IF;
		IF (T_Visu.T_PlcParam.dwActualPage = 110) THEN
			T_Visu.ptrT_ExchgParam^.T_InfoValueCommon.rActualWireFeedPosition:=	T_Station.THardware.TAxisToolFeeder.T_LiveValue.lrActualPosition -
																						T_NovRam.T_Data.T_ProcessImageData.T_CalibrationPara.rStartPosToolFeedCalib;
		END_IF;
		IF (T_Visu.T_PlcParam.dwActualPage = 30) THEN
			T_Visu.ptrT_ExchgParam^.T_InfoValueCommon.rActualWireFeedPosition:=	T_Station.THardware.TAxisToolFeeder.T_LiveValue.lrActualPosition;
		END_IF;
		IF (T_Visu.T_PlcParam.dwActualPage = 330) THEN
			T_Visu.ptrT_ExchgParam^.T_InfoValueCommon.rActualWireFeedPosition:=	T_Station.THardware.TAxisToolFeeder.T_LiveValue.lrActualPosition;
		END_IF;
		T_Visu.ptrT_ExchgParam^.T_StationCommon.rActualToolFeederPosition:=T_Station.THardware.TAxisToolFeeder.T_LiveValue.lrActualPosition;
		T_Visu.ptrT_ExchgParam^.T_InfoValueCommon.rActualWireFeedSpeed:=T_Station.THardware.TAxisToolFeeder.T_LiveValue.lrActualVelocity;
	ELSE
		(* On the MicroWire set the Position of the ToolFeed every time when the TeachPage will be activate to zero *)
		IF (T_Visu.T_PlcParam.dwActualPage = 310) AND NOT(xReadActualToolFeedPos) THEN
			rActualToolFeederPosition:=T_Station.THardware.TAxisToolFeeder.T_LiveValue.lrActualPosition;
			xReadActualToolFeedPos:=TRUE;
		END_IF;
		IF (T_Visu.T_PlcParam.dwActualPage <> 310) THEN
			xReadActualToolFeedPos:=FALSE;
		END_IF;
		T_Visu.ptrT_ExchgParam^.T_StationCommon.rActualToolFeederPosition:=T_Station.THardware.TAxisToolFeeder.T_LiveValue.lrActualPosition - rActualToolFeederPosition;
		(* On the MicroWire set the Position of the ToolFeed every time when the Reference Page will be activate to zero *)
		IF (T_Visu.T_PlcParam.dwActualPage = 30) AND NOT(xReadActualToolFeedPos1) THEN
			rActualToolFeederPosition1:=T_Station.THardware.TAxisToolFeeder.T_LiveValue.lrActualPosition;
			xReadActualToolFeedPos1:=TRUE;
		END_IF;
		IF (T_Visu.T_PlcParam.dwActualPage <> 30) THEN
			xReadActualToolFeedPos1:=FALSE;
		END_IF;
		IF (T_Visu.T_PlcParam.dwActualPage = 30) THEN
			T_Visu.ptrT_ExchgParam^.T_InfoValueCommon.rActualWireFeedPosition:=T_Station.THardware.TAxisToolFeeder.T_LiveValue.lrActualPosition - rActualToolFeederPosition1;
			T_Visu.ptrT_ExchgParam^.T_InfoValueCommon.rActualWireFeedSpeed:=T_Station.THardware.TAxisToolFeeder.T_LiveValue.lrActualVelocity;
		END_IF;
	END_IF;
	T_Visu.ptrT_ExchgParam^.T_InfoValueCommon.rActualGrindAxisPosition:=T_Station.THardware.TAxisGrindFeeder.T_LiveValue.lrActualPosition;
	T_Visu.ptrT_ExchgParam^.T_InfoValueCommon.rActualGrindAxisSpeed:=T_Station.THardware.TAxisGrindFeeder.T_LiveValue.lrActualVelocity;
	T_Visu.ptrT_ExchgParam^.T_StationCommon.rActualGrindFeederPosition:=T_Station.THardware.TAxisGrindFeeder.T_LiveValue.lrActualPosition;
	IF (T_Visu.ptrT_ExchgParam^.T_TeachIn.iSaveToolFeederPos = 0) THEN
		T_Visu.ptrT_ExchgParam^.T_StationCommon.rOldToolFeederPosition:=0.0;
	END_IF;
	IF (T_Visu.ptrT_ExchgParam^.T_TeachIn.iSaveToolFeederPos = 1) THEN
		T_Visu.ptrT_ExchgParam^.T_StationCommon.rOldToolFeederPosition:=T_NovRam.T_Data.T_ProcessImageData.T_ProcessPara.rStartPosToolFeedAuto;
	END_IF;
	IF (T_Visu.ptrT_ExchgParam^.T_TeachIn.iSaveToolFeederPos = 2) THEN
		T_Visu.ptrT_ExchgParam^.T_StationCommon.rOldToolFeederPosition:=T_NovRam.T_Data.T_ProcessImageData.T_CalibrationPara.rStartPosToolFeedCalib;
	END_IF;
	IF (T_Visu.ptrT_ExchgParam^.T_TeachIn.iSaveToolFeederPos = 3) THEN
		T_Visu.ptrT_ExchgParam^.T_StationCommon.rOldToolFeederPosition:=T_NovRam.T_Data.T_ProcessImageData.T_CalibrationPara.rMeasurePosToolFeedCalib;
	END_IF;
	IF (T_Visu.ptrT_ExchgParam^.T_TeachIn.iSaveToolFeederPos = 4) THEN
		T_Visu.ptrT_ExchgParam^.T_StationCommon.rOldToolFeederPosition:=T_NovRam.T_Data.T_Standard.T_AxisPosition.rLoadPosToolFeedAuto;
	END_IF;
	IF (T_Visu.ptrT_ExchgParam^.T_TeachIn.iSaveGrindFeederPos = 0) THEN
		T_Visu.ptrT_ExchgParam^.T_StationCommon.rOldGrindFeederPosition:=0.0;
	END_IF;
	IF (T_Visu.ptrT_ExchgParam^.T_TeachIn.iSaveGrindFeederPos = 1) THEN
		T_Visu.ptrT_ExchgParam^.T_StationCommon.rOldGrindFeederPosition:=T_NovRam.T_Data.T_ProcessImageData.T_ProcessPara.rToolDiameterProcess;
	END_IF;
	IF (T_Visu.ptrT_ExchgParam^.T_TeachIn.iSaveGrindFeederPos = 2) THEN
		(* Security Position will be calculateted with the settled Tooldiameter plus the Offset *)
		T_Visu.ptrT_ExchgParam^.T_StationCommon.rOldGrindFeederPosition:=	T_NovRam.T_Data.T_ProcessImageData.T_ProcessPara.rToolDiameterProcess +
																		T_NovRam.T_Data.T_ProcessImageData.T_ProcessPara.rSecurityPosGrindFeedProcess;
	END_IF;
	IF (T_Visu.ptrT_ExchgParam^.T_TeachIn.iSaveGrindFeederPos = 3) THEN
		T_Visu.ptrT_ExchgParam^.T_StationCommon.rOldGrindFeederPosition:=T_NovRam.T_Data.T_ProcessImageData.T_PrismPara.rToolDiameterMin;
	END_IF;
	IF (T_Visu.ptrT_ExchgParam^.T_TeachIn.iSaveGrindFeederPos = 4) THEN
		T_Visu.ptrT_ExchgParam^.T_StationCommon.rOldGrindFeederPosition:=T_NovRam.T_Data.T_ProcessImageData.T_PrismPara.rToolDiameterMax + T_NovRam.T_Data.T_Standard.T_TeachINGrindFeeder.rOffsetSWPosEndSwitch;
	END_IF;

(* Monitoring Cylinder value *)
	(* Cyl ToolTension *)
	T_Visu.ptrT_ExchgParam^.T_Cylinder.xToolTension:=T_Station.THardware.TCylToolTension.T_CtrleCyl.T_AnalogCylinder.xActiv;
	IF T_Station.THardware.TCylToolTension.T_CtrleCyl.xStatePosOn THEN T_Visu.ptrT_ExchgParam^.T_Cylinder.bPosToolTension:=T_Visu.ptrT_ExchgParam^.T_Cylinder.bPosToolTension OR 16#1;
		ELSE T_Visu.ptrT_ExchgParam^.T_Cylinder.bPosToolTension:=T_Visu.ptrT_ExchgParam^.T_Cylinder.bPosToolTension AND 16#FE; END_IF
	IF (T_Visu.ptrT_ExchgParam^.T_Cylinder.iSelectToolTensionForce < 2) THEN
		T_Visu.ptrT_ExchgParam^.T_Cylinder.rToSetToolTensionForce:=T_NovRam.T_Data.T_ProcessImageData.T_ProcessPara.rToolTensionProcess;
	END_IF;
	IF (T_Visu.ptrT_ExchgParam^.T_Cylinder.iSelectToolTensionForce > 1) THEN
		T_Visu.ptrT_ExchgParam^.T_Cylinder.rToSetToolTensionForce:=T_NovRam.T_Data.T_Standard.T_Cyl_ToolTension.rForce;
	END_IF;
	(*22.12.2009: KFS	{	 *)
	IF xMicroRodActive THEN
		(* Cyl ToolLeft *)
		T_Visu.ptrT_ExchgParam^.T_Cylinder.xCylToolLeft:=T_Station.THardware.TCylToolLeftActive.T_CtrleCyl.T_Standard.xActivOn;
		IF T_Station.THardware.TCylToolLeftActive.T_CtrleCyl.xStatePosOn THEN T_Visu.ptrT_ExchgParam^.T_Cylinder.bPosCylToolLeft:=T_Visu.ptrT_ExchgParam^.T_Cylinder.bPosCylToolLeft OR 16#1;
			ELSE T_Visu.ptrT_ExchgParam^.T_Cylinder.bPosCylToolLeft:=T_Visu.ptrT_ExchgParam^.T_Cylinder.bPosCylToolLeft AND 16#FE; END_IF
		IF T_Station.THardware.TCylToolLeftActive.T_CtrleCyl.xStatePosOff THEN T_Visu.ptrT_ExchgParam^.T_Cylinder.bPosCylToolLeft:=T_Visu.ptrT_ExchgParam^.T_Cylinder.bPosCylToolLeft OR 16#2;
			ELSE T_Visu.ptrT_ExchgParam^.T_Cylinder.bPosCylToolLeft:=T_Visu.ptrT_ExchgParam^.T_Cylinder.bPosCylToolLeft AND 16#FD; END_IF
		(* Cyl ToolRight *)
		T_Visu.ptrT_ExchgParam^.T_Cylinder.xCylToolRight:=T_Station.THardware.TCylToolRightActive.T_CtrleCyl.T_Standard.xActivOn;
		IF T_Station.THardware.TCylToolRightActive.T_CtrleCyl.xStatePosOn THEN T_Visu.ptrT_ExchgParam^.T_Cylinder.bPosCylToolRight:=T_Visu.ptrT_ExchgParam^.T_Cylinder.bPosCylToolRight OR 16#1;
			ELSE T_Visu.ptrT_ExchgParam^.T_Cylinder.bPosCylToolRight:=T_Visu.ptrT_ExchgParam^.T_Cylinder.bPosCylToolRight AND 16#FE; END_IF
		IF T_Station.THardware.TCylToolRightActive.T_CtrleCyl.xStatePosOff THEN T_Visu.ptrT_ExchgParam^.T_Cylinder.bPosCylToolRight:=T_Visu.ptrT_ExchgParam^.T_Cylinder.bPosCylToolRight OR 16#2;
			ELSE T_Visu.ptrT_ExchgParam^.T_Cylinder.bPosCylToolRight:=T_Visu.ptrT_ExchgParam^.T_Cylinder.bPosCylToolRight AND 16#FD; END_IF
		(* Cyl ToolCenter *)
		T_Visu.ptrT_ExchgParam^.T_Cylinder.xCylToolCenter:=T_Station.THardware.TCylToolCenterActive.T_CtrleCyl.T_Standard.xActivOn;
		IF T_Station.THardware.TCylToolCenterActive.T_CtrleCyl.xStatePosOn THEN T_Visu.ptrT_ExchgParam^.T_Cylinder.bPosCylToolCenter:=T_Visu.ptrT_ExchgParam^.T_Cylinder.bPosCylToolCenter OR 16#1;
			ELSE T_Visu.ptrT_ExchgParam^.T_Cylinder.bPosCylToolCenter:=T_Visu.ptrT_ExchgParam^.T_Cylinder.bPosCylToolCenter AND 16#FE; END_IF
		IF T_Station.THardware.TCylToolCenterActive.T_CtrleCyl.xStatePosOff THEN T_Visu.ptrT_ExchgParam^.T_Cylinder.bPosCylToolCenter:=T_Visu.ptrT_ExchgParam^.T_Cylinder.bPosCylToolCenter OR 16#2;
			ELSE T_Visu.ptrT_ExchgParam^.T_Cylinder.bPosCylToolCenter:=T_Visu.ptrT_ExchgParam^.T_Cylinder.bPosCylToolCenter AND 16#FD; END_IF
		(* Cyl ToolPrismaLeft *)
		T_Visu.ptrT_ExchgParam^.T_Cylinder.xCylToolPrismaLeft:=T_Station.THardware.TCylToolPrismaLeftActive.T_CtrleCyl.T_Standard.xActivOn;
		IF T_Station.THardware.TCylToolPrismaLeftActive.T_CtrleCyl.xStatePosOn THEN T_Visu.ptrT_ExchgParam^.T_Cylinder.bPosCylToolPrismaLeft:=T_Visu.ptrT_ExchgParam^.T_Cylinder.bPosCylToolPrismaLeft OR 16#1;
			ELSE T_Visu.ptrT_ExchgParam^.T_Cylinder.bPosCylToolPrismaLeft:=T_Visu.ptrT_ExchgParam^.T_Cylinder.bPosCylToolPrismaLeft AND 16#FE; END_IF
		IF T_Station.THardware.TCylToolPrismaLeftActive.T_CtrleCyl.xStatePosOff THEN T_Visu.ptrT_ExchgParam^.T_Cylinder.bPosCylToolPrismaLeft:=T_Visu.ptrT_ExchgParam^.T_Cylinder.bPosCylToolPrismaLeft OR 16#2;
			ELSE T_Visu.ptrT_ExchgParam^.T_Cylinder.bPosCylToolPrismaLeft:=T_Visu.ptrT_ExchgParam^.T_Cylinder.bPosCylToolPrismaLeft AND 16#FD; END_IF
		(* Cyl ToolPrismaRight *)
		T_Visu.ptrT_ExchgParam^.T_Cylinder.xCylToolPrismaRight:=T_Station.THardware.TCylToolPrismaRightActive.T_CtrleCyl.T_Standard.xActivOn;
		IF T_Station.THardware.TCylToolPrismaRightActive.T_CtrleCyl.xStatePosOn THEN T_Visu.ptrT_ExchgParam^.T_Cylinder.bPosCylToolPrismalRight:=T_Visu.ptrT_ExchgParam^.T_Cylinder.bPosCylToolPrismalRight OR 16#1;
			ELSE T_Visu.ptrT_ExchgParam^.T_Cylinder.bPosCylToolPrismalRight:=T_Visu.ptrT_ExchgParam^.T_Cylinder.bPosCylToolPrismalRight AND 16#FE; END_IF
		IF T_Station.THardware.TCylToolPrismaRightActive.T_CtrleCyl.xStatePosOff THEN T_Visu.ptrT_ExchgParam^.T_Cylinder.bPosCylToolPrismalRight:=T_Visu.ptrT_ExchgParam^.T_Cylinder.bPosCylToolPrismalRight OR 16#2;
			ELSE T_Visu.ptrT_ExchgParam^.T_Cylinder.bPosCylToolPrismalRight:=T_Visu.ptrT_ExchgParam^.T_Cylinder.bPosCylToolPrismalRight AND 16#FD; END_IF
	END_IF;
	(*22.12.2009: KFS	}	 *)

(* Bt Function panel *)
	(* Fn Bt function panel state *)
	CASE T_Visu.T_PlcParam.dwActualPage OF
	10:			wTmp:=16#0;
				IF T_Visu.ptrT_ExchgParam^.T_StationCommon.T_AutoGeometryPara.xPlungeActivationGeometry THEN wTmp:=wTmp+16#1; ELSE wTmp:=wTmp AND 16#FE; END_IF
				IF T_Visu.ptrT_ExchgParam^.T_StationCommon.T_AutoGeometryPara.xDisplaceActivationGeometry THEN wTmp:=wTmp+16#2; ELSE wTmp:=wTmp AND 16#FD; END_IF
				IF T_Visu.ptrT_ExchgParam^.T_Cylinder.xToolTension THEN wTmp:=wTmp+16#4; ELSE wTmp:=wTmp AND 16#FB; END_IF
				IF T_Visu.ptrT_ExchgParam^.T_StationCommon.T_AutoGeometryPara.xWarmUp THEN wTmp:=wTmp+16#20; ELSE wTmp:=wTmp AND 16#DF; END_IF
				xTmp:=	T_Station.THardware.TAxisToolLeft.T_CtrleSingle.xPower AND
						((T_Station.THardware.TAxisToolCenter.T_CtrleSingle.xPower AND xMicroRodActive) OR NOT(xMicroRodActive)) AND
						T_Station.THardware.TAxisToolRight.T_CtrleSingle.xPower AND
						T_Station.THardware.TAxisToolFeeder.T_CtrleSingle.xPower AND
						T_Station.THardware.TAxisGrindFeeder.T_CtrleSingle.xPower;
				IF xTmp THEN wTmp:=wTmp+16#8; ELSE wTmp:=wTmp AND 16#F7; END_IF
	20:			wTmp:=16#0;
				IF T_Visu.ptrT_ExchgParam^.T_StationCommon.T_AutoGroovePara.xPlungeActivationGroove THEN wTmp:=wTmp+16#1; ELSE wTmp:=wTmp AND 16#FE; END_IF
				IF T_Visu.ptrT_ExchgParam^.T_StationCommon.T_AutoGroovePara.xDisplaceActivationGroove THEN wTmp:=wTmp+16#2; ELSE wTmp:=wTmp AND 16#FD; END_IF
				IF T_Visu.ptrT_ExchgParam^.T_Cylinder.xToolTension THEN wTmp:=wTmp+16#4; ELSE wTmp:=wTmp AND 16#FB; END_IF
				IF T_Visu.ptrT_ExchgParam^.T_StationCommon.T_AutoGroovePara.xBlockGrindFeeder THEN wTmp:=wTmp+16#20; ELSE wTmp:=wTmp AND 16#DF; END_IF
	30:			wTmp:=16#0;
				IF T_Visu.ptrT_ExchgParam^.T_Cylinder.xToolTension THEN wTmp:=wTmp+16#4; ELSE wTmp:=wTmp AND 16#FB; END_IF
				xTmp:=	T_Station.THardware.TAxisToolLeft.T_CtrleSingle.xPower AND
						((T_Station.THardware.TAxisToolCenter.T_CtrleSingle.xPower AND xMicroRodActive) OR NOT(xMicroRodActive)) AND
						T_Station.THardware.TAxisToolRight.T_CtrleSingle.xPower AND
						T_Station.THardware.TAxisToolFeeder.T_CtrleSingle.xPower AND
						T_Station.THardware.TAxisGrindFeeder.T_CtrleSingle.xPower;
				IF xTmp THEN wTmp:=wTmp+16#8; ELSE wTmp:=wTmp AND 16#F7; END_IF
	110:			wTmp:=16#0;
				IF T_Visu.ptrT_ExchgParam^.T_StationCommon.T_CalibrationPara.xPlungeActivationCalib THEN wTmp:=wTmp+16#1; ELSE wTmp:=wTmp AND 16#FE; END_IF
				IF T_Visu.ptrT_ExchgParam^.T_StationCommon.T_CalibrationPara.xDisplaceActivationCalib THEN wTmp:=wTmp+16#2; ELSE wTmp:=wTmp AND 16#FD; END_IF
				IF T_Visu.ptrT_ExchgParam^.T_Cylinder.xToolTension THEN wTmp:=wTmp+16#4; ELSE wTmp:=wTmp AND 16#FB; END_IF
	220:			wTmp:=16#0;
				IF T_Visu.ptrT_ExchgParam^.T_Cylinder.xToolTension THEN wTmp:=wTmp+16#4; ELSE wTmp:=wTmp AND 16#FB; END_IF
	310:			wTmp:=16#0;
				IF T_Visu.ptrT_ExchgParam^.T_Cylinder.xToolTension THEN wTmp:=wTmp+16#10; ELSE wTmp:=wTmp AND 16#EF; END_IF
	330:			wTmp:=16#0;
				IF T_Visu.ptrT_ExchgParam^.T_Cylinder.xToolTension THEN wTmp:=wTmp+16#10; ELSE wTmp:=wTmp AND 16#EF; END_IF
				xTmp:=	T_Station.THardware.TAxisToolLeft.T_CtrleSingle.xPower AND
						((T_Station.THardware.TAxisToolCenter.T_CtrleSingle.xPower AND xMicroRodActive) OR NOT(xMicroRodActive)) AND
						T_Station.THardware.TAxisToolRight.T_CtrleSingle.xPower AND
						T_Station.THardware.TAxisToolFeeder.T_CtrleSingle.xPower AND
						T_Station.THardware.TAxisGrindFeeder.T_CtrleSingle.xPower;
				IF xTmp THEN wTmp:=wTmp+16#1; ELSE wTmp:=wTmp AND 16#FE; END_IF
	ELSE wTmp:=16#0;
	END_CASE
	T_Visu.ptrT_ExchgParam^.T_BtFunctionPanel.wState:=wTmp;

(* Monitoring ToolTorque *)
	IF (T_Visu.T_PlcParam.dwActualPage = 220) THEN
		T_Visu.ptrT_ExchgParam^.T_InfoValueCommon.rActualToolLeftTorque:=T_Station.THardware.TAxisToolLeft.T_LiveValue.uiActualTorque;
		T_Visu.ptrT_ExchgParam^.T_InfoValueCommon.rActualToolRightTorque:=T_Station.THardware.TAxisToolRight.T_LiveValue.uiActualTorque;
		T_Visu.ptrT_ExchgParam^.T_InfoValueCommon.rActualToolCenterTorque:=T_Station.THardware.TAxisToolCenter.T_LiveValue.uiActualTorque;
		FBCalcTorqueToolLeft(	xStart:=TRUE,
								uiActualTorque:= T_Station.THardware.TAxisToolLeft.T_LiveValue.uiActualTorque,
								uiZeroTorque:=uiToolLeftZeroTorque,
								iStepCalc:= 100);
		FBCalcTorqueToolCenter(	xStart:=TRUE,
								uiActualTorque:= T_Station.THardware.TAxisToolCenter.T_LiveValue.uiActualTorque,
								uiZeroTorque:=uiToolCenterZeroTorque,
								iStepCalc:= 100);
		FBCalcTorqueToolRight(	xStart:=TRUE,
								uiActualTorque:= T_Station.THardware.TAxisToolRight.T_LiveValue.uiActualTorque,
								uiZeroTorque:=uiToolRightZeroTorque,
								iStepCalc:= 100);
		T_Visu.ptrT_ExchgParam^.T_InfoValueCommon.rCalculToolLeftTorque:=FBCalcTorqueToolLeft.uiCalcTorque;
		T_Visu.ptrT_ExchgParam^.T_InfoValueCommon.rCalculToolCenterTorque:=FBCalcTorqueToolCenter.uiCalcTorque;
		T_Visu.ptrT_ExchgParam^.T_InfoValueCommon.rCalculToolRightTorque:=FBCalcTorqueToolRight.uiCalcTorque;
	ELSE
		FBCalcTorqueToolLeft(	xStart:=FALSE);
		FBCalcTorqueToolCenter(	xStart:=FALSE);
		FBCalcTorqueToolRight(	xStart:=FALSE);
	END_IF;

(* Monitoring Max ToolRotation Speed *)
	IF xMicroRodActive THEN
		T_Visu.ptrT_ExchgParam^.T_StationCommon.rMaxSpeedToolRotation:=1200.0;
	ELSE
		T_Visu.ptrT_ExchgParam^.T_StationCommon.rMaxSpeedToolRotation:=500.0;
	END_IF;

(* Monitoring AutoGeometry or AutoGroove *)
	IF (T_Visu.T_PlcParam.dwActualPage = 10) OR (T_Visu.T_PlcParam.dwActualPage = 20) THEN
		xPart1:=xPart2:=xPart3:=xPart4:=FALSE;
		rToolTotalLength:=0.0;
		IF T_Visu.ptrT_ExchgParam^.T_GeometryCommon.T_Geometry.axActiveSection[1] THEN
			xPart1:=TRUE;
			T_Visu.ptrT_ExchgParam^.T_InfoValueCommon.arStartDiameter[1]:=T_Visu.ptrT_ExchgParam^.T_GeometryCommon.T_Geometry.arStartDiameter[1];
			T_Visu.ptrT_ExchgParam^.T_InfoValueCommon.arEndDiameter[1]:=T_Visu.ptrT_ExchgParam^.T_GeometryCommon.T_Geometry.arEndDiameter[1];
			rToolTotalLength:=rToolTotalLength + T_Visu.ptrT_ExchgParam^.T_GeometryCommon.T_Geometry.arSectionLength[1];
			IF T_Visu.ptrT_ExchgParam^.T_GeometryCommon.T_Geometry.axActiveSection[2] THEN
				xPart2:=TRUE;
				T_Visu.ptrT_ExchgParam^.T_InfoValueCommon.arStartDiameter[2]:=T_Visu.ptrT_ExchgParam^.T_GeometryCommon.T_Geometry.arStartDiameter[2];
				T_Visu.ptrT_ExchgParam^.T_InfoValueCommon.arEndDiameter[2]:=T_Visu.ptrT_ExchgParam^.T_GeometryCommon.T_Geometry.arEndDiameter[2];
				rToolTotalLength:=rToolTotalLength + T_Visu.ptrT_ExchgParam^.T_GeometryCommon.T_Geometry.arSectionLength[2];
				IF T_Visu.ptrT_ExchgParam^.T_GeometryCommon.T_Geometry.axActiveSection[3] THEN
					xPart3:=TRUE;
					T_Visu.ptrT_ExchgParam^.T_InfoValueCommon.arStartDiameter[3]:=T_Visu.ptrT_ExchgParam^.T_GeometryCommon.T_Geometry.arStartDiameter[3];
					T_Visu.ptrT_ExchgParam^.T_InfoValueCommon.arEndDiameter[3]:=T_Visu.ptrT_ExchgParam^.T_GeometryCommon.T_Geometry.arEndDiameter[3];
					rToolTotalLength:=rToolTotalLength + T_Visu.ptrT_ExchgParam^.T_GeometryCommon.T_Geometry.arSectionLength[3];
					IF T_Visu.ptrT_ExchgParam^.T_GeometryCommon.T_Geometry.axActiveSection[4] THEN
						xPart4:=TRUE;
						T_Visu.ptrT_ExchgParam^.T_InfoValueCommon.arStartDiameter[4]:=T_Visu.ptrT_ExchgParam^.T_GeometryCommon.T_Geometry.arStartDiameter[4];
						T_Visu.ptrT_ExchgParam^.T_InfoValueCommon.arEndDiameter[4]:=T_Visu.ptrT_ExchgParam^.T_GeometryCommon.T_Geometry.arEndDiameter[4];
						rToolTotalLength:=rToolTotalLength + T_Visu.ptrT_ExchgParam^.T_GeometryCommon.T_Geometry.arSectionLength[4];
					END_IF;
				END_IF;
			END_IF;
		ELSIF T_Visu.ptrT_ExchgParam^.T_GeometryCommon.T_Geometry.axActiveSection[2] THEN
			xPart2:=TRUE;
			T_Visu.ptrT_ExchgParam^.T_InfoValueCommon.arStartDiameter[1]:=T_Visu.ptrT_ExchgParam^.T_GeometryCommon.T_Geometry.arStartDiameter[2];
			T_Visu.ptrT_ExchgParam^.T_InfoValueCommon.arEndDiameter[1]:=T_Visu.ptrT_ExchgParam^.T_GeometryCommon.T_Geometry.arEndDiameter[2];
			rToolTotalLength:=rToolTotalLength + T_Visu.ptrT_ExchgParam^.T_GeometryCommon.T_Geometry.arSectionLength[2];
			IF T_Visu.ptrT_ExchgParam^.T_GeometryCommon.T_Geometry.axActiveSection[3] THEN
				xPart3:=TRUE;
				T_Visu.ptrT_ExchgParam^.T_InfoValueCommon.arStartDiameter[2]:=T_Visu.ptrT_ExchgParam^.T_GeometryCommon.T_Geometry.arStartDiameter[3];
				T_Visu.ptrT_ExchgParam^.T_InfoValueCommon.arEndDiameter[2]:=T_Visu.ptrT_ExchgParam^.T_GeometryCommon.T_Geometry.arEndDiameter[3];
				rToolTotalLength:=rToolTotalLength + T_Visu.ptrT_ExchgParam^.T_GeometryCommon.T_Geometry.arSectionLength[3];
				IF T_Visu.ptrT_ExchgParam^.T_GeometryCommon.T_Geometry.axActiveSection[4] THEN
					xPart4:=TRUE;
					T_Visu.ptrT_ExchgParam^.T_InfoValueCommon.arStartDiameter[3]:=T_Visu.ptrT_ExchgParam^.T_GeometryCommon.T_Geometry.arStartDiameter[4];
					T_Visu.ptrT_ExchgParam^.T_InfoValueCommon.arEndDiameter[3]:=T_Visu.ptrT_ExchgParam^.T_GeometryCommon.T_Geometry.arEndDiameter[4];
					rToolTotalLength:=rToolTotalLength + T_Visu.ptrT_ExchgParam^.T_GeometryCommon.T_Geometry.arSectionLength[4];
				END_IF;
			END_IF;
		ELSIF T_Visu.ptrT_ExchgParam^.T_GeometryCommon.T_Geometry.axActiveSection[3] THEN
			xPart3:=TRUE;
			T_Visu.ptrT_ExchgParam^.T_InfoValueCommon.arStartDiameter[1]:=T_Visu.ptrT_ExchgParam^.T_GeometryCommon.T_Geometry.arStartDiameter[3];
			T_Visu.ptrT_ExchgParam^.T_InfoValueCommon.arEndDiameter[1]:=T_Visu.ptrT_ExchgParam^.T_GeometryCommon.T_Geometry.arEndDiameter[3];
			rToolTotalLength:=rToolTotalLength + T_Visu.ptrT_ExchgParam^.T_GeometryCommon.T_Geometry.arSectionLength[3];
			IF T_Visu.ptrT_ExchgParam^.T_GeometryCommon.T_Geometry.axActiveSection[4] THEN
				xPart4:=TRUE;
				T_Visu.ptrT_ExchgParam^.T_InfoValueCommon.arStartDiameter[2]:=T_Visu.ptrT_ExchgParam^.T_GeometryCommon.T_Geometry.arStartDiameter[4];
				T_Visu.ptrT_ExchgParam^.T_InfoValueCommon.arEndDiameter[2]:=T_Visu.ptrT_ExchgParam^.T_GeometryCommon.T_Geometry.arEndDiameter[4];
				rToolTotalLength:=rToolTotalLength + T_Visu.ptrT_ExchgParam^.T_GeometryCommon.T_Geometry.arSectionLength[4];
			END_IF;
		ELSIF T_Visu.ptrT_ExchgParam^.T_GeometryCommon.T_Geometry.axActiveSection[4] THEN
			xPart4:=TRUE;
			T_Visu.ptrT_ExchgParam^.T_InfoValueCommon.arStartDiameter[1]:=T_Visu.ptrT_ExchgParam^.T_GeometryCommon.T_Geometry.arStartDiameter[4];
			T_Visu.ptrT_ExchgParam^.T_InfoValueCommon.arEndDiameter[1]:=T_Visu.ptrT_ExchgParam^.T_GeometryCommon.T_Geometry.arEndDiameter[4];
			rToolTotalLength:=rToolTotalLength + T_Visu.ptrT_ExchgParam^.T_GeometryCommon.T_Geometry.arSectionLength[4];
		ELSE
			FOR ii:=1 TO 4 DO
				T_Visu.ptrT_ExchgParam^.T_InfoValueCommon.arStartDiameter[ii]:=0;
				T_Visu.ptrT_ExchgParam^.T_InfoValueCommon.arEndDiameter[ii]:=0;
			END_FOR;
		END_IF;
		iPartActive:=0;
		IF xPart1 THEN iPartActive:=iPartActive + 1; END_IF;
		IF xPart2 THEN iPartActive:=iPartActive + 1; END_IF;
		IF xPart3 THEN iPartActive:=iPartActive + 1; END_IF;
		IF xPart4 THEN iPartActive:=iPartActive + 1; END_IF;
		IF (iPartActive > 0) THEN
			FOR ii:=4 TO (iPartActive + 1) BY -1 DO
				T_Visu.ptrT_ExchgParam^.T_InfoValueCommon.arStartDiameter[ii]:=0;
				T_Visu.ptrT_ExchgParam^.T_InfoValueCommon.arEndDiameter[ii]:=0;
			END_FOR;
		END_IF;
		T_Visu.ptrT_ExchgParam^.T_InfoValueCommon.iTotalCountDownCycle:=T_NovRAM.T_Data.T_ProcessImageData.T_AutoGeometryPara.iCycleGeometry;
		T_Visu.ptrT_ExchgParam^.T_InfoValueCommon.iTotalCountDownPlungeCycle:=T_Station.T_WorkTool.iTotalCountDownPlungeCycle;
		T_Visu.ptrT_ExchgParam^.T_InfoValueCommon.iTotalCountDownGrooveCycle:=T_NovRAM.T_Data.T_ProcessImageData.T_AutoGroovePara.iNumberOfGrooves;
		T_Visu.ptrT_ExchgParam^.T_InfoValueCommon.rToolDiameter:=T_NovRAM.T_Data.T_ProcessImageData.T_ProcessPara.rToolDiameterProcess;
		T_Visu.ptrT_ExchgParam^.T_InfoValueCommon.rToolTotalLength:=rToolTotalLength * 10.0;	(* umwandeln von cm in mm *)
		IF (T_Visu.T_PlcParam.dwActualPage = 10) THEN
			IF T_NovRAM.T_Data.T_ProcessImageData.T_AutoGeometryPara.xPlungeActivationGeometry THEN
				T_Visu.ptrT_ExchgParam^.T_InfoValueCommon.rToolTotalLength:=T_Visu.ptrT_ExchgParam^.T_InfoValueCommon.rToolTotalLength + T_NovRAM.T_Data.T_ProcessImageData.T_AutoGeometryPara.rPlungeLengthToolFeedGeometry;
			END_IF;
			IF T_NovRAM.T_Data.T_ProcessImageData.T_AutoGeometryPara.xDisplaceActivationGeometry THEN
				T_Visu.ptrT_ExchgParam^.T_InfoValueCommon.rToolTotalLength:=T_Visu.ptrT_ExchgParam^.T_InfoValueCommon.rToolTotalLength + T_NovRAM.T_Data.T_ProcessImageData.T_AutoGeometryPara.rDisplaceLengthToolFeedGeometry;
			END_IF;
		END_IF;
		IF (T_Visu.T_PlcParam.dwActualPage = 20) THEN
			IF T_NovRAM.T_Data.T_ProcessImageData.T_AutoGroovePara.xPlungeActivationGroove AND NOT(T_NovRAM.T_Data.T_ProcessImageData.T_AutoGroovePara.xBlockGrindFeeder) THEN
				T_Visu.ptrT_ExchgParam^.T_InfoValueCommon.rToolTotalLength:=T_Visu.ptrT_ExchgParam^.T_InfoValueCommon.rToolTotalLength + T_NovRAM.T_Data.T_ProcessImageData.T_AutoGroovePara.rPlungeLengthToolFeedGroove;
			END_IF;
			IF T_NovRAM.T_Data.T_ProcessImageData.T_AutoGroovePara.xDisplaceActivationGroove THEN
				T_Visu.ptrT_ExchgParam^.T_InfoValueCommon.rToolTotalLength:=T_Visu.ptrT_ExchgParam^.T_InfoValueCommon.rToolTotalLength + T_NovRAM.T_Data.T_ProcessImageData.T_AutoGroovePara.rDisplaceLengthToolFeedGroove;
			END_IF;
		END_IF;
	ELSE
		T_Visu.ptrT_ExchgParam^.T_InfoValueCommon.iCountDownCycle:=1;
		T_Visu.ptrT_ExchgParam^.T_InfoValueCommon.iCountDownPlungeCycle:=1;
		T_Visu.ptrT_ExchgParam^.T_InfoValueCommon.iCountDownGrooveCycle:=1;
	END_IF;

